Universal Robots URScript: 2024DragonThinMarker_v7.script

def P2024DragonThinMarker_v7():
  step_count_72c97e26_6cb8_45e0_928f_f3c530a1ae50 = 0.0
  thread Step_Counter_Thread_41fc0684_b974_431a_b44c_1ae3c598adf5():
    while (True):
      step_count_72c97e26_6cb8_45e0_928f_f3c530a1ae50 = step_count_72c97e26_6cb8_45e0_928f_f3c530a1ae50 + 1.0
      sync()
    end
  end
  run Step_Counter_Thread_41fc0684_b974_431a_b44c_1ae3c598adf5()
  set_gravity([0.0, 0.0, 9.82])
  set_tcp(p[0.0,0.0,0.0,0.0,0.0,0.0])
  set_standard_analog_input_domain(0, 1)
  set_standard_analog_input_domain(1, 1)
  set_tool_analog_input_domain(0, 1)
  set_tool_analog_input_domain(1, 1)
  set_analog_outputdomain(0, 0)
  set_analog_outputdomain(1, 0)
  set_input_actions_to_default()
  set_target_payload(1.070000, [0.002000, 0.003000, 0.057000], [0.001723, 0.001723, 0.001723, 0.000000, 0.000000, 0.000000])
  set_safety_mode_transition_hardness(1)
  set_tool_communication(True, 1000000, 2, 1, 1.5, 3.5)
  set_tool_output_mode(0)
  set_tool_digital_output_mode(0, 1)
  set_tool_digital_output_mode(1, 1)
  set_tool_voltage(0)
  global Plane_1=p[-0.700006141123905,1.3454883874109249E-6,0.3910559577028425,-1.2089868272251132,-1.2089999932245832,1.20858562628424]
  global Plane_2=p[0.0,0.0,0.0,0.0,0.0,0.0]
  global Point_1=p[0.6913645118948067,-0.12399382748223003,0.49223711947071,-1.2983729986843258,1.1259514972191385,-1.2203503861141718]
  $ 1 "Robot Program"
  $ 2 "Script: polyu_fai_chun_2024.script"
  def Machining1():
    # Default parameters:
    global speed_ms = 0.3
    global speed_rads = 0.75
    global accel_mss = 3
    global accel_radss = 1.2
    global blend_radius_m = 0.001

    # Add subprograms here
    # Start of main program
    # Program generated by RoboDK v5.6.5 for UR10e on 12/01/2024 18:22:17
    # Using nominal kinematics.
    blend_radius_m = 0.000
    speed_ms = 1.000
    # set_reference(p[0.335000, -0.149886, -0.015500, 0.000000, 0.000000, 0.000000])
    set_tcp(p[0.000000, 0.000000, 0.252000, 0.000000, 0.000000, 0.000000])
    # Show Tool
    movej([0.073712, -1.005472, -2.512389, -1.194528, 1.570796, 1.644508],accel_radss,speed_rads,0,blend_radius_m)
    movel([0.073712, -1.005472, -2.512389, -1.194528, 1.570796, 1.644508],accel_mss,speed_ms,0,blend_radius_m)
    # Splitting Linear movement in 6 (instruction 7: MoveL 3)
    movel([0.073712, -1.023685, -2.537003, -1.151700, 1.570796, 1.644508],accel_mss,speed_ms,0,blend_radius_m)
    movel([0.073712, -1.044503, -2.561079, -1.106807, 1.570796, 1.644508],accel_mss,speed_ms,0,blend_radius_m)
    movel([0.073712, -1.068168, -2.584569, -1.059651, 1.570796, 1.644508],accel_mss,speed_ms,0,blend_radius_m)
    movel([0.073712, -1.094942, -2.607420, -1.010026, 1.570796, 1.644508],accel_mss,speed_ms,0,blend_radius_m)
    movel([0.073712, -1.125104, -2.629569, -0.957717, 1.570796, 1.644508],accel_mss,speed_ms,0,blend_radius_m)
    movel([0.073712, -1.158943, -2.650939, -0.902506, 1.570796, 1.644508],accel_mss,speed_ms,0,blend_radius_m)
    movel([0.073712, -1.158943, -2.650939, -0.902506, 1.570796, 1.644508],accel_mss,speed_ms,0,blend_radius_m)
    speed_ms = 1.000
    movel([0.073712, -1.158943, -2.650939, -0.902506, 1.570796, 1.644508],accel_mss,speed_ms,0,blend_radius_m)
    movel([0.073712, -1.158943, -2.650939, -0.902506, 1.570796, 1.644508],accel_mss,speed_ms,0,blend_radius_m)
    movel([0.073712, -1.158943, -2.650939, -0.902506, 1.570796, 1.644508],accel_mss,speed_ms,0,blend_radius_m)
    speed_ms = 0.005
    movel([0.073712, -1.118787, -2.625199, -0.968404, 1.570796, 1.644508],accel_mss,speed_ms,0,blend_radius_m)
    speed_ms = 1.000
    movel([0.073712, -1.158943, -2.650939, -0.902506, 1.570796, 1.644508],accel_mss,speed_ms,0,blend_radius_m)
    speed_ms = 0.040
    movel([0.073712, -1.158943, -2.650939, -0.902506, 1.570796, 1.644508],accel_mss,speed_ms,0,blend_radius_m)
    speed_ms = 1.000
    movel([0.073712, -1.158943, -2.650939, -0.902506, 1.570796, 1.644508],accel_mss,speed_ms,0,blend_radius_m)
    # Splitting Linear movement in 4 (instruction 21: MoveL 12)
    movel([0.101880, -1.181857, -2.640286, -0.890246, 1.570796, 1.672676],accel_mss,speed_ms,0,blend_radius_m)
    movel([0.128207, -1.205564, -2.628681, -0.878144, 1.570796, 1.699004],accel_mss,speed_ms,0,blend_radius_m)
    movel([0.152802, -1.229857, -2.616150, -0.866382, 1.570796, 1.723598],accel_mss,speed_ms,0,blend_radius_m)
    movel([0.175774, -1.254553, -2.602722, -0.855114, 1.570796, 1.746570],accel_mss,speed_ms,0,blend_radius_m)
    speed_ms = 0.005
    movel([0.175774, -1.298704, -2.625119, -0.788567, 1.570796, 1.746570],accel_mss,speed_ms,0,blend_radius_m)
    speed_ms = 0.025
    movel([0.175467, -1.296515, -2.626415, -0.789459, 1.570796, 1.746263],accel_mss,speed_ms,0,blend_radius_m)
    movel([0.175132, -1.295590, -2.626961, -0.789837, 1.570796, 1.745929],accel_mss,speed_ms,0,blend_radius_m)
    movel([0.174656, -1.294762, -2.627449, -0.790178, 1.570796, 1.745452],accel_mss,speed_ms,0,blend_radius_m)
    movel([0.174050, -1.294049, -2.627869, -0.790471, 1.570796, 1.744846],accel_mss,speed_ms,0,blend_radius_m)
    movel([0.173318, -1.293452, -2.628219, -0.790718, 1.570796, 1.744114],accel_mss,speed_ms,0,blend_radius_m)
    movel([0.172433, -1.292952, -2.628513, -0.790925, 1.570796, 1.743230],accel_mss,speed_ms,0,blend_radius_m)
    movel([0.171452, -1.292568, -2.628738, -0.791083, 1.570796, 1.742248],accel_mss,speed_ms,0,blend_radius_m)
    movel([0.169238, -1.292109, -2.629007, -0.791274, 1.570796, 1.740034],accel_mss,speed_ms,0,blend_radius_m)
    movel([0.166824, -1.292044, -2.629045, -0.791300, 1.570796, 1.737621],accel_mss,speed_ms,0,blend_radius_m)
    movel([0.164077, -1.292380, -2.628848, -0.791161, 1.570796, 1.734873],accel_mss,speed_ms,0,blend_radius_m)
    movel([0.160852, -1.293136, -2.628405, -0.790848, 1.570796, 1.731649],accel_mss,speed_ms,0,blend_radius_m)
    movel([0.158343, -1.293899, -2.627957, -0.790533, 1.570796, 1.729139],accel_mss,speed_ms,0,blend_radius_m)
    movel([0.156195, -1.294698, -2.627487, -0.790204, 1.570796, 1.726992],accel_mss,speed_ms,0,blend_radius_m)
    movel([0.154013, -1.295690, -2.626903, -0.789797, 1.570796, 1.724809],accel_mss,speed_ms,0,blend_radius_m)
    movel([0.151400, -1.297044, -2.626103, -0.789243, 1.570796, 1.722196],accel_mss,speed_ms,0,blend_radius_m)
    movel([0.148354, -1.298788, -2.625069, -0.788532, 1.570796, 1.719150],accel_mss,speed_ms,0,blend_radius_m)
    movel([0.140219, -1.303870, -2.622034, -0.786485, 1.570796, 1.711015],accel_mss,speed_ms,0,blend_radius_m)
    movel([0.140032, -1.304046, -2.621928, -0.786415, 1.570796, 1.710829],accel_mss,speed_ms,0,blend_radius_m)
    movel([0.139940, -1.304251, -2.621805, -0.786333, 1.570796, 1.710737],accel_mss,speed_ms,0,blend_radius_m)
    movel([0.140046, -1.304840, -2.621451, -0.786098, 1.570796, 1.710842],accel_mss,speed_ms,0,blend_radius_m)
    movel([0.143328, -1.309440, -2.618669, -0.784280, 1.570796, 1.714124],accel_mss,speed_ms,0,blend_radius_m)
    movel([0.145350, -1.311978, -2.617122, -0.783289, 1.570796, 1.716147],accel_mss,speed_ms,0,blend_radius_m)
    movel([0.153033, -1.320929, -2.611599, -0.779860, 1.570796, 1.723829],accel_mss,speed_ms,0,blend_radius_m)
    movel([0.157376, -1.325880, -2.608499, -0.778010, 1.570796, 1.728172],accel_mss,speed_ms,0,blend_radius_m)
    movel([0.160651, -1.329420, -2.606262, -0.776707, 1.570796, 1.731447],accel_mss,speed_ms,0,blend_radius_m)
    movel([0.161108, -1.329847, -2.605991, -0.776551, 1.570796, 1.731904],accel_mss,speed_ms,0,blend_radius_m)
    movel([0.161761, -1.330342, -2.605676, -0.776371, 1.570796, 1.732557],accel_mss,speed_ms,0,blend_radius_m)
    movel([0.162354, -1.330373, -2.605656, -0.776359, 1.570796, 1.733150],accel_mss,speed_ms,0,blend_radius_m)
    movel([0.162959, -1.330023, -2.605879, -0.776487, 1.570796, 1.733755],accel_mss,speed_ms,0,blend_radius_m)
    movel([0.163738, -1.329104, -2.606462, -0.776823, 1.570796, 1.734534],accel_mss,speed_ms,0,blend_radius_m)
    movel([0.165104, -1.327071, -2.607748, -0.777570, 1.570796, 1.735901],accel_mss,speed_ms,0,blend_radius_m)
    movel([0.167659, -1.322835, -2.610409, -0.779144, 1.570796, 1.738455],accel_mss,speed_ms,0,blend_radius_m)
    movel([0.169919, -1.318408, -2.613166, -0.780815, 1.570796, 1.740716],accel_mss,speed_ms,0,blend_radius_m)
    movel([0.171903, -1.313743, -2.616042, -0.782604, 1.570796, 1.742699],accel_mss,speed_ms,0,blend_radius_m)
    movel([0.173625, -1.308797, -2.619060, -0.784532, 1.570796, 1.744421],accel_mss,speed_ms,0,blend_radius_m)
    movel([0.174404, -1.306055, -2.620719, -0.785615, 1.570796, 1.745200],accel_mss,speed_ms,0,blend_radius_m)
    movel([0.175649, -1.300261, -2.624193, -0.787936, 1.570796, 1.746445],accel_mss,speed_ms,0,blend_radius_m)
    movel([0.175774, -1.298704, -2.625119, -0.788567, 1.570796, 1.746570],accel_mss,speed_ms,0,blend_radius_m)
    movel([0.175467, -1.296515, -2.626415, -0.789459, 1.570796, 1.746263],accel_mss,speed_ms,0,blend_radius_m)
    speed_ms = 0.005
    movel([0.175467, -1.287281, -2.622040, -0.803067, 1.570796, 1.746263],accel_mss,speed_ms,0,blend_radius_m)
    speed_ms = 0.040
    movel([0.174810, -1.299280, -2.614952, -0.798157, 1.570796, 1.745606],accel_mss,speed_ms,0,blend_radius_m)
    speed_ms = 0.005
    movel([0.174810, -1.308444, -2.619274, -0.784671, 1.570796, 1.745606],accel_mss,speed_ms,0,blend_radius_m)
    speed_ms = 0.025
    movel([0.172959, -1.313681, -2.616080, -0.782628, 1.570796, 1.743756],accel_mss,speed_ms,0,blend_radius_m)
    movel([0.171021, -1.318273, -2.613249, -0.780867, 1.570796, 1.741817],accel_mss,speed_ms,0,blend_radius_m)
    movel([0.168851, -1.322542, -2.610593, -0.779254, 1.570796, 1.739648],accel_mss,speed_ms,0,blend_radius_m)
    movel([0.166314, -1.326792, -2.607924, -0.777673, 1.570796, 1.737110],accel_mss,speed_ms,0,blend_radius_m)
    movel([0.163959, -1.330191, -2.605772, -0.776426, 1.570796, 1.734756],accel_mss,speed_ms,0,blend_radius_m)
    movel([0.163273, -1.330890, -2.605328, -0.776171, 1.570796, 1.734070],accel_mss,speed_ms,0,blend_radius_m)
    movel([0.162439, -1.331386, -2.605012, -0.775991, 1.570796, 1.733235],accel_mss,speed_ms,0,blend_radius_m)
    movel([0.161654, -1.331560, -2.604902, -0.775928, 1.570796, 1.732450],accel_mss,speed_ms,0,blend_radius_m)
    movel([0.161027, -1.331383, -2.605014, -0.775992, 1.570796, 1.731824],accel_mss,speed_ms,0,blend_radius_m)
    movel([0.159182, -1.329800, -2.606021, -0.776568, 1.570796, 1.729978],accel_mss,speed_ms,0,blend_radius_m)
    movel([0.154933, -1.325131, -2.608970, -0.778288, 1.570796, 1.725729],accel_mss,speed_ms,0,blend_radius_m)
    movel([0.149543, -1.318950, -2.612830, -0.780609, 1.570796, 1.720340],accel_mss,speed_ms,0,blend_radius_m)
    movel([0.144364, -1.312895, -2.616561, -0.782932, 1.570796, 1.715160],accel_mss,speed_ms,0,blend_radius_m)
    movel([0.141237, -1.308969, -2.618955, -0.784465, 1.570796, 1.712033],accel_mss,speed_ms,0,blend_radius_m)
    movel([0.139694, -1.306790, -2.620275, -0.785324, 1.570796, 1.710491],accel_mss,speed_ms,0,blend_radius_m)
    movel([0.138982, -1.305403, -2.621112, -0.785874, 1.570796, 1.709778],accel_mss,speed_ms,0,blend_radius_m)
    movel([0.138836, -1.304410, -2.621710, -0.786270, 1.570796, 1.709632],accel_mss,speed_ms,0,blend_radius_m)
    movel([0.138954, -1.304019, -2.621945, -0.786426, 1.570796, 1.709750],accel_mss,speed_ms,0,blend_radius_m)
    movel([0.139242, -1.303642, -2.622171, -0.786576, 1.570796, 1.710039],accel_mss,speed_ms,0,blend_radius_m)
    movel([0.139895, -1.303121, -2.622483, -0.786785, 1.570796, 1.710691],accel_mss,speed_ms,0,blend_radius_m)
    movel([0.145279, -1.299642, -2.624561, -0.788186, 1.570796, 1.716076],accel_mss,speed_ms,0,blend_radius_m)
    movel([0.147733, -1.298138, -2.625454, -0.788797, 1.570796, 1.718530],accel_mss,speed_ms,0,blend_radius_m)
    movel([0.150828, -1.296376, -2.626497, -0.789515, 1.570796, 1.721624],accel_mss,speed_ms,0,blend_radius_m)
    movel([0.153961, -1.294776, -2.627441, -0.790172, 1.570796, 1.724758],accel_mss,speed_ms,0,blend_radius_m)
    movel([0.156801, -1.293517, -2.628181, -0.790691, 1.570796, 1.727598],accel_mss,speed_ms,0,blend_radius_m)
    movel([0.159642, -1.292475, -2.628792, -0.791122, 1.570796, 1.730438],accel_mss,speed_ms,0,blend_radius_m)
    movel([0.162247, -1.291733, -2.629227, -0.791430, 1.570796, 1.733043],accel_mss,speed_ms,0,blend_radius_m)
    movel([0.164801, -1.291232, -2.629519, -0.791638, 1.570796, 1.735598],accel_mss,speed_ms,0,blend_radius_m)
    movel([0.167190, -1.290996, -2.629657, -0.791736, 1.570796, 1.737986],accel_mss,speed_ms,0,blend_radius_m)
    movel([0.169469, -1.291023, -2.629641, -0.791725, 1.570796, 1.740266],accel_mss,speed_ms,0,blend_radius_m)
    movel([0.171128, -1.291248, -2.629510, -0.791631, 1.570796, 1.741924],accel_mss,speed_ms,0,blend_radius_m)
    movel([0.172657, -1.291674, -2.629261, -0.791454, 1.570796, 1.743454],accel_mss,speed_ms,0,blend_radius_m)
    movel([0.173914, -1.292270, -2.628912, -0.791207, 1.570796, 1.744711],accel_mss,speed_ms,0,blend_radius_m)
    movel([0.174977, -1.293079, -2.628438, -0.790872, 1.570796, 1.745773],accel_mss,speed_ms,0,blend_radius_m)
    movel([0.175808, -1.294073, -2.627854, -0.790461, 1.570796, 1.746605],accel_mss,speed_ms,0,blend_radius_m)
    movel([0.176410, -1.295244, -2.627165, -0.789980, 1.570796, 1.747207],accel_mss,speed_ms,0,blend_radius_m)
    movel([0.176810, -1.296630, -2.626347, -0.789412, 1.570796, 1.747606],accel_mss,speed_ms,0,blend_radius_m)
    movel([0.176990, -1.298135, -2.625456, -0.788798, 1.570796, 1.747786],accel_mss,speed_ms,0,blend_radius_m)
    movel([0.176880, -1.299644, -2.624560, -0.788185, 1.570796, 1.747676],accel_mss,speed_ms,0,blend_radius_m)
    movel([0.176287, -1.302678, -2.622749, -0.786962, 1.570796, 1.747084],accel_mss,speed_ms,0,blend_radius_m)
    movel([0.175547, -1.305881, -2.620824, -0.785684, 1.570796, 1.746344],accel_mss,speed_ms,0,blend_radius_m)
    movel([0.174810, -1.308444, -2.619274, -0.784671, 1.570796, 1.745606],accel_mss,speed_ms,0,blend_radius_m)
    movel([0.173912, -1.310987, -2.617727, -0.783675, 1.570796, 1.744708],accel_mss,speed_ms,0,blend_radius_m)
    speed_ms = 0.005
    movel([0.173912, -1.301837, -2.613417, -0.797134, 1.570796, 1.744708],accel_mss,speed_ms,0,blend_radius_m)
    speed_ms = 0.040
    # Splitting Linear movement in 4 (instruction 117: MoveL 100)
    movel([0.163813, -1.329309, -2.596395, -0.786686, 1.570796, 1.734610],accel_mss,speed_ms,0,blend_radius_m)
    movel([0.154297, -1.355614, -2.579147, -0.777628, 1.570796, 1.725093],accel_mss,speed_ms,0,blend_radius_m)
    movel([0.145312, -1.380862, -2.561692, -0.769834, 1.570796, 1.716108],accel_mss,speed_ms,0,blend_radius_m)
    movel([0.136812, -1.405151, -2.544044, -0.763194, 1.570796, 1.707609],accel_mss,speed_ms,0,blend_radius_m)
    speed_ms = 0.005
    movel([0.136812, -1.413611, -2.547901, -0.750877, 1.570796, 1.707609],accel_mss,speed_ms,0,blend_radius_m)
    speed_ms = 0.025
    movel([0.136960, -1.413086, -2.548297, -0.751006, 1.570796, 1.707756],accel_mss,speed_ms,0,blend_radius_m)
    movel([0.137280, -1.410569, -2.550188, -0.751632, 1.570796, 1.708076],accel_mss,speed_ms,0,blend_radius_m)
    movel([0.137084, -1.408675, -2.551604, -0.752109, 1.570796, 1.707880],accel_mss,speed_ms,0,blend_radius_m)
    movel([0.136478, -1.406567, -2.553175, -0.752647, 1.570796, 1.707274],accel_mss,speed_ms,0,blend_radius_m)
    movel([0.135486, -1.404266, -2.554882, -0.753241, 1.570796, 1.706282],accel_mss,speed_ms,0,blend_radius_m)
    movel([0.134091, -1.401787, -2.556712, -0.753889, 1.570796, 1.704888],accel_mss,speed_ms,0,blend_radius_m)
    movel([0.133438, -1.400815, -2.557428, -0.754146, 1.570796, 1.704235],accel_mss,speed_ms,0,blend_radius_m)
    movel([0.132951, -1.400309, -2.557799, -0.754280, 1.570796, 1.703748],accel_mss,speed_ms,0,blend_radius_m)
    movel([0.132501, -1.400110, -2.557946, -0.754333, 1.570796, 1.703298],accel_mss,speed_ms,0,blend_radius_m)
    movel([0.132010, -1.400164, -2.557906, -0.754319, 1.570796, 1.702806],accel_mss,speed_ms,0,blend_radius_m)
    movel([0.131521, -1.400467, -2.557683, -0.754238, 1.570796, 1.702317],accel_mss,speed_ms,0,blend_radius_m)
    movel([0.131266, -1.400883, -2.557378, -0.754128, 1.570796, 1.702062],accel_mss,speed_ms,0,blend_radius_m)
    movel([0.131373, -1.401180, -2.557160, -0.754050, 1.570796, 1.702169],accel_mss,speed_ms,0,blend_radius_m)
    movel([0.132162, -1.401260, -2.557101, -0.754029, 1.570796, 1.702958],accel_mss,speed_ms,0,blend_radius_m)
    movel([0.132555, -1.401611, -2.556842, -0.753936, 1.570796, 1.703352],accel_mss,speed_ms,0,blend_radius_m)
    movel([0.134004, -1.403943, -2.555121, -0.753325, 1.570796, 1.704800],accel_mss,speed_ms,0,blend_radius_m)
    movel([0.135071, -1.406059, -2.553553, -0.752777, 1.570796, 1.705868],accel_mss,speed_ms,0,blend_radius_m)
    movel([0.135785, -1.408024, -2.552090, -0.752275, 1.570796, 1.706581],accel_mss,speed_ms,0,blend_radius_m)
    movel([0.136159, -1.409851, -2.550725, -0.751812, 1.570796, 1.706955],accel_mss,speed_ms,0,blend_radius_m)
    movel([0.136189, -1.411547, -2.549454, -0.751388, 1.570796, 1.706985],accel_mss,speed_ms,0,blend_radius_m)
    movel([0.136087, -1.412720, -2.548572, -0.751097, 1.570796, 1.706884],accel_mss,speed_ms,0,blend_radius_m)
    movel([0.135567, -1.411763, -2.549291, -0.751334, 1.570796, 1.706364],accel_mss,speed_ms,0,blend_radius_m)
    movel([0.134960, -1.410840, -2.549984, -0.751564, 1.570796, 1.705756],accel_mss,speed_ms,0,blend_radius_m)
    movel([0.134201, -1.410029, -2.550592, -0.751768, 1.570796, 1.704998],accel_mss,speed_ms,0,blend_radius_m)
    movel([0.133183, -1.409207, -2.551207, -0.751975, 1.570796, 1.703979],accel_mss,speed_ms,0,blend_radius_m)
    movel([0.132066, -1.408483, -2.551748, -0.752158, 1.570796, 1.702862],accel_mss,speed_ms,0,blend_radius_m)
    movel([0.130773, -1.407814, -2.552247, -0.752328, 1.570796, 1.701569],accel_mss,speed_ms,0,blend_radius_m)
    movel([0.129389, -1.407256, -2.552662, -0.752470, 1.570796, 1.700185],accel_mss,speed_ms,0,blend_radius_m)
    movel([0.127928, -1.406809, -2.552995, -0.752585, 1.570796, 1.698724],accel_mss,speed_ms,0,blend_radius_m)
    movel([0.126392, -1.406478, -2.553242, -0.752670, 1.570796, 1.697188],accel_mss,speed_ms,0,blend_radius_m)
    movel([0.124687, -1.406237, -2.553421, -0.752732, 1.570796, 1.695483],accel_mss,speed_ms,0,blend_radius_m)
    movel([0.123487, -1.406221, -2.553432, -0.752735, 1.570796, 1.694283],accel_mss,speed_ms,0,blend_radius_m)
    movel([0.122540, -1.406414, -2.553289, -0.752686, 1.570796, 1.693336],accel_mss,speed_ms,0,blend_radius_m)
    movel([0.121683, -1.406830, -2.552980, -0.752579, 1.570796, 1.692479],accel_mss,speed_ms,0,blend_radius_m)
    movel([0.121218, -1.407199, -2.552705, -0.752485, 1.570796, 1.692014],accel_mss,speed_ms,0,blend_radius_m)
    movel([0.120891, -1.407598, -2.552408, -0.752383, 1.570796, 1.691687],accel_mss,speed_ms,0,blend_radius_m)
    movel([0.120677, -1.408078, -2.552050, -0.752261, 1.570796, 1.691473],accel_mss,speed_ms,0,blend_radius_m)
    movel([0.120519, -1.409292, -2.551143, -0.751953, 1.570796, 1.691315],accel_mss,speed_ms,0,blend_radius_m)
    movel([0.120597, -1.410164, -2.550491, -0.751734, 1.570796, 1.691393],accel_mss,speed_ms,0,blend_radius_m)
    movel([0.120924, -1.411776, -2.549282, -0.751331, 1.570796, 1.691721],accel_mss,speed_ms,0,blend_radius_m)
    movel([0.120137, -1.411178, -2.549731, -0.751480, 1.570796, 1.690933],accel_mss,speed_ms,0,blend_radius_m)
    movel([0.119142, -1.410325, -2.550371, -0.751693, 1.570796, 1.689938],accel_mss,speed_ms,0,blend_radius_m)
    movel([0.118017, -1.409589, -2.550922, -0.751879, 1.570796, 1.688813],accel_mss,speed_ms,0,blend_radius_m)
    movel([0.116588, -1.408871, -2.551458, -0.752060, 1.570796, 1.687384],accel_mss,speed_ms,0,blend_radius_m)
    movel([0.114638, -1.408066, -2.552059, -0.752264, 1.570796, 1.685434],accel_mss,speed_ms,0,blend_radius_m)
    movel([0.110959, -1.406603, -2.553148, -0.752637, 1.570796, 1.681756],accel_mss,speed_ms,0,blend_radius_m)
    movel([0.108642, -1.405547, -2.553933, -0.752909, 1.570796, 1.679439],accel_mss,speed_ms,0,blend_radius_m)
    movel([0.106996, -1.404575, -2.554653, -0.753160, 1.570796, 1.677792],accel_mss,speed_ms,0,blend_radius_m)
    movel([0.105601, -1.403457, -2.555480, -0.753451, 1.570796, 1.676397],accel_mss,speed_ms,0,blend_radius_m)
    movel([0.105049, -1.402986, -2.555828, -0.753574, 1.570796, 1.675845],accel_mss,speed_ms,0,blend_radius_m)
    movel([0.104656, -1.402804, -2.555963, -0.753622, 1.570796, 1.675452],accel_mss,speed_ms,0,blend_radius_m)
    movel([0.104367, -1.402858, -2.555923, -0.753608, 1.570796, 1.675163],accel_mss,speed_ms,0,blend_radius_m)
    movel([0.104133, -1.403095, -2.555748, -0.753546, 1.570796, 1.674929],accel_mss,speed_ms,0,blend_radius_m)
    movel([0.104093, -1.403268, -2.555620, -0.753501, 1.570796, 1.674889],accel_mss,speed_ms,0,blend_radius_m)
    movel([0.104524, -1.406129, -2.553501, -0.752759, 1.570796, 1.675320],accel_mss,speed_ms,0,blend_radius_m)
    movel([0.104631, -1.406790, -2.553009, -0.752590, 1.570796, 1.675427],accel_mss,speed_ms,0,blend_radius_m)
    movel([0.104692, -1.407427, -2.552536, -0.752427, 1.570796, 1.675488],accel_mss,speed_ms,0,blend_radius_m)
    movel([0.102290, -1.405992, -2.553602, -0.752794, 1.570796, 1.673087],accel_mss,speed_ms,0,blend_radius_m)
    movel([0.100620, -1.404841, -2.554457, -0.753092, 1.570796, 1.671417],accel_mss,speed_ms,0,blend_radius_m)
    movel([0.099425, -1.403815, -2.555216, -0.753358, 1.570796, 1.670222],accel_mss,speed_ms,0,blend_radius_m)
    movel([0.098377, -1.402613, -2.556104, -0.753672, 1.570796, 1.669174],accel_mss,speed_ms,0,blend_radius_m)
    movel([0.095814, -1.399011, -2.558752, -0.754627, 1.570796, 1.666610],accel_mss,speed_ms,0,blend_radius_m)
    movel([0.094727, -1.397866, -2.559589, -0.754934, 1.570796, 1.665523],accel_mss,speed_ms,0,blend_radius_m)
    movel([0.093735, -1.397245, -2.560043, -0.755101, 1.570796, 1.664531],accel_mss,speed_ms,0,blend_radius_m)
    movel([0.093259, -1.397104, -2.560145, -0.755139, 1.570796, 1.664056],accel_mss,speed_ms,0,blend_radius_m)
    movel([0.092715, -1.397075, -2.560166, -0.755147, 1.570796, 1.663511],accel_mss,speed_ms,0,blend_radius_m)
    movel([0.092023, -1.397198, -2.560077, -0.755114, 1.570796, 1.662819],accel_mss,speed_ms,0,blend_radius_m)
    movel([0.091298, -1.397494, -2.559861, -0.755034, 1.570796, 1.662095],accel_mss,speed_ms,0,blend_radius_m)
    movel([0.090566, -1.397956, -2.559523, -0.754910, 1.570796, 1.661362],accel_mss,speed_ms,0,blend_radius_m)
    movel([0.089095, -1.399249, -2.558577, -0.754563, 1.570796, 1.659892],accel_mss,speed_ms,0,blend_radius_m)
    movel([0.088807, -1.398175, -2.559363, -0.754851, 1.570796, 1.659604],accel_mss,speed_ms,0,blend_radius_m)
    movel([0.088677, -1.397590, -2.559790, -0.755008, 1.570796, 1.659474],accel_mss,speed_ms,0,blend_radius_m)
    movel([0.086678, -1.390759, -2.564745, -0.756884, 1.570796, 1.657474],accel_mss,speed_ms,0,blend_radius_m)
    movel([0.086361, -1.389318, -2.565782, -0.757289, 1.570796, 1.657158],accel_mss,speed_ms,0,blend_radius_m)
    movel([0.086303, -1.388031, -2.566706, -0.757652, 1.570796, 1.657099],accel_mss,speed_ms,0,blend_radius_m)
    movel([0.086463, -1.385965, -2.568183, -0.758241, 1.570796, 1.657259],accel_mss,speed_ms,0,blend_radius_m)
    movel([0.086845, -1.383220, -2.570135, -0.759033, 1.570796, 1.657641],accel_mss,speed_ms,0,blend_radius_m)
    movel([0.087125, -1.382255, -2.570820, -0.759315, 1.570796, 1.657921],accel_mss,speed_ms,0,blend_radius_m)
    movel([0.088538, -1.378520, -2.573454, -0.760415, 1.570796, 1.659334],accel_mss,speed_ms,0,blend_radius_m)
    movel([0.088847, -1.377865, -2.573914, -0.760610, 1.570796, 1.659643],accel_mss,speed_ms,0,blend_radius_m)
    movel([0.089252, -1.377361, -2.574268, -0.760760, 1.570796, 1.660049],accel_mss,speed_ms,0,blend_radius_m)
    movel([0.089322, -1.377088, -2.574459, -0.760842, 1.570796, 1.660119],accel_mss,speed_ms,0,blend_radius_m)
    movel([0.089228, -1.376863, -2.574617, -0.760909, 1.570796, 1.660025],accel_mss,speed_ms,0,blend_radius_m)
    movel([0.088991, -1.376732, -2.574708, -0.760949, 1.570796, 1.659787],accel_mss,speed_ms,0,blend_radius_m)
    movel([0.088772, -1.376745, -2.574699, -0.760945, 1.570796, 1.659568],accel_mss,speed_ms,0,blend_radius_m)
    movel([0.088542, -1.376869, -2.574612, -0.760908, 1.570796, 1.659338],accel_mss,speed_ms,0,blend_radius_m)
    movel([0.088083, -1.377390, -2.574248, -0.760752, 1.570796, 1.658880],accel_mss,speed_ms,0,blend_radius_m)
    movel([0.087563, -1.378426, -2.573520, -0.760443, 1.570796, 1.658359],accel_mss,speed_ms,0,blend_radius_m)
    movel([0.086135, -1.382410, -2.570710, -0.759269, 1.570796, 1.656932],accel_mss,speed_ms,0,blend_radius_m)
    movel([0.085693, -1.383923, -2.569636, -0.758830, 1.570796, 1.656489],accel_mss,speed_ms,0,blend_radius_m)
    movel([0.085220, -1.386694, -2.567662, -0.758033, 1.570796, 1.656017],accel_mss,speed_ms,0,blend_radius_m)
    movel([0.085156, -1.388244, -2.566553, -0.757592, 1.570796, 1.655952],accel_mss,speed_ms,0,blend_radius_m)
    movel([0.085288, -1.389626, -2.565561, -0.757202, 1.570796, 1.656084],accel_mss,speed_ms,0,blend_radius_m)
    movel([0.085687, -1.391336, -2.564330, -0.756723, 1.570796, 1.656483],accel_mss,speed_ms,0,blend_radius_m)
    movel([0.087127, -1.396101, -2.560877, -0.755411, 1.570796, 1.657923],accel_mss,speed_ms,0,blend_radius_m)
    movel([0.087508, -1.397558, -2.559814, -0.755017, 1.570796, 1.658304],accel_mss,speed_ms,0,blend_radius_m)
    movel([0.088079, -1.400709, -2.557506, -0.754174, 1.570796, 1.658875],accel_mss,speed_ms,0,blend_radius_m)
    movel([0.088230, -1.401088, -2.557227, -0.754074, 1.570796, 1.659026],accel_mss,speed_ms,0,blend_radius_m)
    movel([0.088515, -1.401157, -2.557177, -0.754056, 1.570796, 1.659311],accel_mss,speed_ms,0,blend_radius_m)
    movel([0.088888, -1.400924, -2.557347, -0.754117, 1.570796, 1.659684],accel_mss,speed_ms,0,blend_radius_m)
    movel([0.089305, -1.400387, -2.557742, -0.754260, 1.570796, 1.660101],accel_mss,speed_ms,0,blend_radius_m)
    movel([0.089783, -1.399740, -2.558217, -0.754432, 1.570796, 1.660580],accel_mss,speed_ms,0,blend_radius_m)
    movel([0.090394, -1.399084, -2.558698, -0.754607, 1.570796, 1.661191],accel_mss,speed_ms,0,blend_radius_m)
    movel([0.091027, -1.398524, -2.559108, -0.754757, 1.570796, 1.661823],accel_mss,speed_ms,0,blend_radius_m)
    movel([0.091557, -1.398188, -2.559353, -0.754847, 1.570796, 1.662354],accel_mss,speed_ms,0,blend_radius_m)
    movel([0.092171, -1.398032, -2.559468, -0.754889, 1.570796, 1.662968],accel_mss,speed_ms,0,blend_radius_m)
    movel([0.092861, -1.398118, -2.559405, -0.754866, 1.570796, 1.663658],accel_mss,speed_ms,0,blend_radius_m)
    movel([0.093562, -1.398429, -2.559178, -0.754783, 1.570796, 1.664359],accel_mss,speed_ms,0,blend_radius_m)
    movel([0.094200, -1.398945, -2.558800, -0.754644, 1.570796, 1.664996],accel_mss,speed_ms,0,blend_radius_m)
    movel([0.094561, -1.399351, -2.558502, -0.754536, 1.570796, 1.665357],accel_mss,speed_ms,0,blend_radius_m)
    movel([0.098013, -1.404105, -2.555001, -0.753283, 1.570796, 1.668809],accel_mss,speed_ms,0,blend_radius_m)
    movel([0.098347, -1.404499, -2.554710, -0.753180, 1.570796, 1.669143],accel_mss,speed_ms,0,blend_radius_m)
    movel([0.099589, -1.405494, -2.553973, -0.752923, 1.570796, 1.670385],accel_mss,speed_ms,0,blend_radius_m)
    movel([0.100597, -1.406207, -2.553443, -0.752739, 1.570796, 1.671393],accel_mss,speed_ms,0,blend_radius_m)
    movel([0.105149, -1.409357, -2.551095, -0.751937, 1.570796, 1.675945],accel_mss,speed_ms,0,blend_radius_m)
    movel([0.106031, -1.410013, -2.550605, -0.751772, 1.570796, 1.676827],accel_mss,speed_ms,0,blend_radius_m)
    movel([0.106225, -1.410030, -2.550591, -0.751767, 1.570796, 1.677021],accel_mss,speed_ms,0,blend_radius_m)
    movel([0.106437, -1.409903, -2.550687, -0.751800, 1.570796, 1.677233],accel_mss,speed_ms,0,blend_radius_m)
    movel([0.106593, -1.409667, -2.550863, -0.751859, 1.570796, 1.677389],accel_mss,speed_ms,0,blend_radius_m)
    movel([0.106611, -1.409441, -2.551033, -0.751916, 1.570796, 1.677408],accel_mss,speed_ms,0,blend_radius_m)
    movel([0.105600, -1.405987, -2.553606, -0.752796, 1.570796, 1.676396],accel_mss,speed_ms,0,blend_radius_m)
    movel([0.105382, -1.404992, -2.554345, -0.753053, 1.570796, 1.676178],accel_mss,speed_ms,0,blend_radius_m)
    movel([0.107701, -1.406321, -2.553358, -0.752710, 1.570796, 1.678497],accel_mss,speed_ms,0,blend_radius_m)
    movel([0.109036, -1.406958, -2.552884, -0.752547, 1.570796, 1.679832],accel_mss,speed_ms,0,blend_radius_m)
    movel([0.112944, -1.408534, -2.551710, -0.752145, 1.570796, 1.683740],accel_mss,speed_ms,0,blend_radius_m)
    movel([0.115927, -1.409742, -2.550807, -0.751840, 1.570796, 1.686724],accel_mss,speed_ms,0,blend_radius_m)
    movel([0.117594, -1.410633, -2.550139, -0.751616, 1.570796, 1.688391],accel_mss,speed_ms,0,blend_radius_m)
    movel([0.119035, -1.411772, -2.549285, -0.751332, 1.570796, 1.689831],accel_mss,speed_ms,0,blend_radius_m)
    movel([0.121575, -1.414285, -2.547393, -0.750712, 1.570796, 1.692371],accel_mss,speed_ms,0,blend_radius_m)
    movel([0.121884, -1.414519, -2.547215, -0.750654, 1.570796, 1.692680],accel_mss,speed_ms,0,blend_radius_m)
    movel([0.122364, -1.414644, -2.547121, -0.750624, 1.570796, 1.693160],accel_mss,speed_ms,0,blend_radius_m)
    movel([0.122659, -1.414449, -2.547268, -0.750671, 1.570796, 1.693456],accel_mss,speed_ms,0,blend_radius_m)
    movel([0.122786, -1.414128, -2.547511, -0.750750, 1.570796, 1.693583],accel_mss,speed_ms,0,blend_radius_m)
    movel([0.122715, -1.413570, -2.547932, -0.750887, 1.570796, 1.693512],accel_mss,speed_ms,0,blend_radius_m)
    movel([0.121659, -1.410088, -2.550548, -0.751753, 1.570796, 1.692455],accel_mss,speed_ms,0,blend_radius_m)
    movel([0.121446, -1.409090, -2.551295, -0.752004, 1.570796, 1.692242],accel_mss,speed_ms,0,blend_radius_m)
    movel([0.121439, -1.408575, -2.551679, -0.752135, 1.570796, 1.692235],accel_mss,speed_ms,0,blend_radius_m)
    movel([0.121484, -1.408388, -2.551819, -0.752182, 1.570796, 1.692280],accel_mss,speed_ms,0,blend_radius_m)
    movel([0.121829, -1.407746, -2.552297, -0.752345, 1.570796, 1.692625],accel_mss,speed_ms,0,blend_radius_m)
    movel([0.122077, -1.407507, -2.552476, -0.752406, 1.570796, 1.692873],accel_mss,speed_ms,0,blend_radius_m)
    movel([0.122378, -1.407341, -2.552599, -0.752449, 1.570796, 1.693174],accel_mss,speed_ms,0,blend_radius_m)
    movel([0.123206, -1.407142, -2.552748, -0.752500, 1.570796, 1.694002],accel_mss,speed_ms,0,blend_radius_m)
    movel([0.124336, -1.407146, -2.552745, -0.752499, 1.570796, 1.695133],accel_mss,speed_ms,0,blend_radius_m)
    movel([0.125835, -1.407372, -2.552576, -0.752441, 1.570796, 1.696631],accel_mss,speed_ms,0,blend_radius_m)
    movel([0.127408, -1.407740, -2.552302, -0.752347, 1.570796, 1.698205],accel_mss,speed_ms,0,blend_radius_m)
    movel([0.128900, -1.408223, -2.551942, -0.752224, 1.570796, 1.699697],accel_mss,speed_ms,0,blend_radius_m)
    movel([0.130280, -1.408803, -2.551509, -0.752077, 1.570796, 1.701076],accel_mss,speed_ms,0,blend_radius_m)
    movel([0.131564, -1.409495, -2.550992, -0.751902, 1.570796, 1.702360],accel_mss,speed_ms,0,blend_radius_m)
    movel([0.132655, -1.410231, -2.550441, -0.751717, 1.570796, 1.703451],accel_mss,speed_ms,0,blend_radius_m)
    movel([0.133637, -1.411071, -2.549812, -0.751507, 1.570796, 1.704434],accel_mss,speed_ms,0,blend_radius_m)
    movel([0.134359, -1.411893, -2.549194, -0.751302, 1.570796, 1.705155],accel_mss,speed_ms,0,blend_radius_m)
    movel([0.134925, -1.412833, -2.548487, -0.751069, 1.570796, 1.705721],accel_mss,speed_ms,0,blend_radius_m)
    movel([0.135624, -1.413985, -2.547619, -0.750785, 1.570796, 1.706420],accel_mss,speed_ms,0,blend_radius_m)
    movel([0.135916, -1.414180, -2.547472, -0.750737, 1.570796, 1.706712],accel_mss,speed_ms,0,blend_radius_m)
    movel([0.136439, -1.414124, -2.547514, -0.750751, 1.570796, 1.707235],accel_mss,speed_ms,0,blend_radius_m)
    movel([0.136587, -1.414019, -2.547593, -0.750777, 1.570796, 1.707383],accel_mss,speed_ms,0,blend_radius_m)
    movel([0.136812, -1.413611, -2.547901, -0.750877, 1.570796, 1.707609],accel_mss,speed_ms,0,blend_radius_m)
    movel([0.136960, -1.413086, -2.548297, -0.751006, 1.570796, 1.707756],accel_mss,speed_ms,0,blend_radius_m)
    movel([0.137159, -1.411521, -2.549473, -0.751394, 1.570796, 1.707955],accel_mss,speed_ms,0,blend_radius_m)
    speed_ms = 0.005
    movel([0.137159, -1.403046, -2.545607, -0.763736, 1.570796, 1.707955],accel_mss,speed_ms,0,blend_radius_m)
    speed_ms = 0.040
    # Splitting Linear movement in 2 (instruction 283: MoveL 262)
    movel([0.174820, -1.398287, -2.549118, -0.764984, 1.570796, 1.745617],accel_mss,speed_ms,0,blend_radius_m)
    movel([0.212258, -1.394754, -2.551703, -0.765932, 1.570796, 1.783055],accel_mss,speed_ms,0,blend_radius_m)
    speed_ms = 0.005
    movel([0.212258, -1.403290, -2.555604, -0.753495, 1.570796, 1.783055],accel_mss,speed_ms,0,blend_radius_m)
    speed_ms = 0.025
    movel([0.212995, -1.402513, -2.556178, -0.753699, 1.570796, 1.783791],accel_mss,speed_ms,0,blend_radius_m)
    movel([0.213276, -1.402201, -2.556407, -0.753780, 1.570796, 1.784073],accel_mss,speed_ms,0,blend_radius_m)
    movel([0.213298, -1.401947, -2.556595, -0.753847, 1.570796, 1.784095],accel_mss,speed_ms,0,blend_radius_m)
    movel([0.213229, -1.401814, -2.556693, -0.753882, 1.570796, 1.784026],accel_mss,speed_ms,0,blend_radius_m)
    movel([0.212929, -1.401746, -2.556743, -0.753900, 1.570796, 1.783725],accel_mss,speed_ms,0,blend_radius_m)
    movel([0.212539, -1.401942, -2.556598, -0.753848, 1.570796, 1.783336],accel_mss,speed_ms,0,blend_radius_m)
    movel([0.211824, -1.402619, -2.556099, -0.753671, 1.570796, 1.782621],accel_mss,speed_ms,0,blend_radius_m)
    movel([0.210769, -1.403737, -2.555273, -0.753378, 1.570796, 1.781565],accel_mss,speed_ms,0,blend_radius_m)
    movel([0.205843, -1.409184, -2.551224, -0.751981, 1.570796, 1.776640],accel_mss,speed_ms,0,blend_radius_m)
    movel([0.204956, -1.410043, -2.550582, -0.751764, 1.570796, 1.775752],accel_mss,speed_ms,0,blend_radius_m)
    movel([0.203263, -1.411446, -2.549530, -0.751413, 1.570796, 1.774059],accel_mss,speed_ms,0,blend_radius_m)
    movel([0.203180, -1.411391, -2.549571, -0.751427, 1.570796, 1.773976],accel_mss,speed_ms,0,blend_radius_m)
    movel([0.204405, -1.409407, -2.551058, -0.751924, 1.570796, 1.775201],accel_mss,speed_ms,0,blend_radius_m)
    movel([0.204693, -1.408783, -2.551524, -0.752082, 1.570796, 1.775490],accel_mss,speed_ms,0,blend_radius_m)
    movel([0.205056, -1.407571, -2.552428, -0.752390, 1.570796, 1.775853],accel_mss,speed_ms,0,blend_radius_m)
    movel([0.205078, -1.407327, -2.552610, -0.752452, 1.570796, 1.775875],accel_mss,speed_ms,0,blend_radius_m)
    movel([0.204845, -1.407180, -2.552720, -0.752490, 1.570796, 1.775641],accel_mss,speed_ms,0,blend_radius_m)
    movel([0.204649, -1.407237, -2.552677, -0.752475, 1.570796, 1.775445],accel_mss,speed_ms,0,blend_radius_m)
    movel([0.204084, -1.407646, -2.552372, -0.752371, 1.570796, 1.774880],accel_mss,speed_ms,0,blend_radius_m)
    movel([0.203703, -1.408009, -2.552101, -0.752278, 1.570796, 1.774499],accel_mss,speed_ms,0,blend_radius_m)
    movel([0.202377, -1.409088, -2.551296, -0.752005, 1.570796, 1.773173],accel_mss,speed_ms,0,blend_radius_m)
    movel([0.200783, -1.409954, -2.550648, -0.751787, 1.570796, 1.771579],accel_mss,speed_ms,0,blend_radius_m)
    movel([0.198815, -1.410647, -2.550129, -0.751613, 1.570796, 1.769612],accel_mss,speed_ms,0,blend_radius_m)
    movel([0.196342, -1.411216, -2.549702, -0.751470, 1.570796, 1.767138],accel_mss,speed_ms,0,blend_radius_m)
    movel([0.193574, -1.411606, -2.549409, -0.751373, 1.570796, 1.764370],accel_mss,speed_ms,0,blend_radius_m)
    movel([0.192481, -1.411670, -2.549362, -0.751357, 1.570796, 1.763278],accel_mss,speed_ms,0,blend_radius_m)
    movel([0.191968, -1.411589, -2.549422, -0.751377, 1.570796, 1.762764],accel_mss,speed_ms,0,blend_radius_m)
    movel([0.193125, -1.410815, -2.550003, -0.751571, 1.570796, 1.763921],accel_mss,speed_ms,0,blend_radius_m)
    movel([0.194094, -1.410188, -2.550473, -0.751728, 1.570796, 1.764890],accel_mss,speed_ms,0,blend_radius_m)
    movel([0.196326, -1.408364, -2.551836, -0.752188, 1.570796, 1.767122],accel_mss,speed_ms,0,blend_radius_m)
    movel([0.196574, -1.407967, -2.552133, -0.752289, 1.570796, 1.767371],accel_mss,speed_ms,0,blend_radius_m)
    movel([0.196504, -1.407757, -2.552290, -0.752343, 1.570796, 1.767301],accel_mss,speed_ms,0,blend_radius_m)
    movel([0.196205, -1.407640, -2.552376, -0.752372, 1.570796, 1.767001],accel_mss,speed_ms,0,blend_radius_m)
    movel([0.194383, -1.407610, -2.552399, -0.752380, 1.570796, 1.765179],accel_mss,speed_ms,0,blend_radius_m)
    movel([0.191988, -1.407594, -2.552411, -0.752384, 1.570796, 1.762784],accel_mss,speed_ms,0,blend_radius_m)
    movel([0.189879, -1.407394, -2.552560, -0.752435, 1.570796, 1.760675],accel_mss,speed_ms,0,blend_radius_m)
    movel([0.188178, -1.407036, -2.552827, -0.752527, 1.570796, 1.758974],accel_mss,speed_ms,0,blend_radius_m)
    movel([0.187061, -1.406523, -2.553208, -0.752658, 1.570796, 1.757858],accel_mss,speed_ms,0,blend_radius_m)
    movel([0.186560, -1.406179, -2.553464, -0.752746, 1.570796, 1.757356],accel_mss,speed_ms,0,blend_radius_m)
    movel([0.188628, -1.405758, -2.553777, -0.752855, 1.570796, 1.759424],accel_mss,speed_ms,0,blend_radius_m)
    movel([0.189090, -1.405630, -2.553872, -0.752888, 1.570796, 1.759886],accel_mss,speed_ms,0,blend_radius_m)
    movel([0.189607, -1.405360, -2.554072, -0.752957, 1.570796, 1.760404],accel_mss,speed_ms,0,blend_radius_m)
    movel([0.189781, -1.405074, -2.554284, -0.753031, 1.570796, 1.760578],accel_mss,speed_ms,0,blend_radius_m)
    movel([0.189749, -1.404838, -2.554459, -0.753092, 1.570796, 1.760546],accel_mss,speed_ms,0,blend_radius_m)
    movel([0.189456, -1.404622, -2.554619, -0.753148, 1.570796, 1.760252],accel_mss,speed_ms,0,blend_radius_m)
    movel([0.187133, -1.403654, -2.555335, -0.753400, 1.570796, 1.757929],accel_mss,speed_ms,0,blend_radius_m)
    movel([0.186609, -1.403384, -2.555534, -0.753470, 1.570796, 1.757405],accel_mss,speed_ms,0,blend_radius_m)
    movel([0.184440, -1.401938, -2.556601, -0.753850, 1.570796, 1.755236],accel_mss,speed_ms,0,blend_radius_m)
    movel([0.183283, -1.401048, -2.557256, -0.754084, 1.570796, 1.754079],accel_mss,speed_ms,0,blend_radius_m)
    movel([0.183316, -1.400879, -2.557381, -0.754129, 1.570796, 1.754112],accel_mss,speed_ms,0,blend_radius_m)
    movel([0.185288, -1.400773, -2.557459, -0.754157, 1.570796, 1.756084],accel_mss,speed_ms,0,blend_radius_m)
    movel([0.185716, -1.400735, -2.557486, -0.754167, 1.570796, 1.756513],accel_mss,speed_ms,0,blend_radius_m)
    movel([0.186580, -1.400524, -2.557642, -0.754223, 1.570796, 1.757376],accel_mss,speed_ms,0,blend_radius_m)
    movel([0.186686, -1.400404, -2.557730, -0.754255, 1.570796, 1.757482],accel_mss,speed_ms,0,blend_radius_m)
    movel([0.186743, -1.400027, -2.558007, -0.754355, 1.570796, 1.757539],accel_mss,speed_ms,0,blend_radius_m)
    movel([0.186632, -1.399840, -2.558143, -0.754405, 1.570796, 1.757428],accel_mss,speed_ms,0,blend_radius_m)
    movel([0.186087, -1.399438, -2.558439, -0.754512, 1.570796, 1.756883],accel_mss,speed_ms,0,blend_radius_m)
    movel([0.185288, -1.398908, -2.558827, -0.754654, 1.570796, 1.756085],accel_mss,speed_ms,0,blend_radius_m)
    movel([0.183948, -1.397503, -2.559855, -0.755032, 1.570796, 1.754744],accel_mss,speed_ms,0,blend_radius_m)
    movel([0.183403, -1.396649, -2.560478, -0.755263, 1.570796, 1.754199],accel_mss,speed_ms,0,blend_radius_m)
    movel([0.182615, -1.394728, -2.561875, -0.755786, 1.570796, 1.753411],accel_mss,speed_ms,0,blend_radius_m)
    movel([0.182409, -1.393739, -2.562593, -0.756058, 1.570796, 1.753206],accel_mss,speed_ms,0,blend_radius_m)
    movel([0.182291, -1.392006, -2.563846, -0.756537, 1.570796, 1.753087],accel_mss,speed_ms,0,blend_radius_m)
    movel([0.182169, -1.391624, -2.564122, -0.756643, 1.570796, 1.752965],accel_mss,speed_ms,0,blend_radius_m)
    movel([0.181958, -1.391488, -2.564220, -0.756681, 1.570796, 1.752755],accel_mss,speed_ms,0,blend_radius_m)
    movel([0.181659, -1.391545, -2.564179, -0.756665, 1.570796, 1.752455],accel_mss,speed_ms,0,blend_radius_m)
    movel([0.181400, -1.391841, -2.563966, -0.756583, 1.570796, 1.752196],accel_mss,speed_ms,0,blend_radius_m)
    movel([0.181291, -1.392472, -2.563509, -0.756407, 1.570796, 1.752087],accel_mss,speed_ms,0,blend_radius_m)
    movel([0.181467, -1.394567, -2.561992, -0.755830, 1.570796, 1.752263],accel_mss,speed_ms,0,blend_radius_m)
    movel([0.181772, -1.395809, -2.561089, -0.755491, 1.570796, 1.752569],accel_mss,speed_ms,0,blend_radius_m)
    movel([0.182255, -1.396984, -2.560233, -0.755172, 1.570796, 1.753052],accel_mss,speed_ms,0,blend_radius_m)
    movel([0.182893, -1.398044, -2.559459, -0.754886, 1.570796, 1.753689],accel_mss,speed_ms,0,blend_radius_m)
    movel([0.183660, -1.398936, -2.558807, -0.754647, 1.570796, 1.754457],accel_mss,speed_ms,0,blend_radius_m)
    movel([0.184310, -1.399597, -2.558322, -0.754470, 1.570796, 1.755106],accel_mss,speed_ms,0,blend_radius_m)
    movel([0.184284, -1.399801, -2.558173, -0.754416, 1.570796, 1.755080],accel_mss,speed_ms,0,blend_radius_m)
    movel([0.184058, -1.399908, -2.558094, -0.754387, 1.570796, 1.754854],accel_mss,speed_ms,0,blend_radius_m)
    movel([0.182268, -1.399637, -2.558293, -0.754459, 1.570796, 1.753064],accel_mss,speed_ms,0,blend_radius_m)
    movel([0.181785, -1.399641, -2.558290, -0.754458, 1.570796, 1.752582],accel_mss,speed_ms,0,blend_radius_m)
    movel([0.181463, -1.399746, -2.558213, -0.754430, 1.570796, 1.752259],accel_mss,speed_ms,0,blend_radius_m)
    movel([0.181244, -1.399951, -2.558063, -0.754376, 1.570796, 1.752041],accel_mss,speed_ms,0,blend_radius_m)
    movel([0.181142, -1.400289, -2.557814, -0.754286, 1.570796, 1.751939],accel_mss,speed_ms,0,blend_radius_m)
    movel([0.181245, -1.400557, -2.557618, -0.754215, 1.570796, 1.752041],accel_mss,speed_ms,0,blend_radius_m)
    movel([0.182830, -1.402051, -2.556518, -0.753820, 1.570796, 1.753626],accel_mss,speed_ms,0,blend_radius_m)
    movel([0.184632, -1.403489, -2.555457, -0.753443, 1.570796, 1.755428],accel_mss,speed_ms,0,blend_radius_m)
    movel([0.186344, -1.404506, -2.554705, -0.753178, 1.570796, 1.757140],accel_mss,speed_ms,0,blend_radius_m)
    movel([0.187606, -1.405119, -2.554250, -0.753020, 1.570796, 1.758402],accel_mss,speed_ms,0,blend_radius_m)
    movel([0.185027, -1.405403, -2.554040, -0.752946, 1.570796, 1.755823],accel_mss,speed_ms,0,blend_radius_m)
    movel([0.184789, -1.405518, -2.553955, -0.752917, 1.570796, 1.755586],accel_mss,speed_ms,0,blend_radius_m)
    movel([0.184643, -1.405700, -2.553819, -0.752870, 1.570796, 1.755439],accel_mss,speed_ms,0,blend_radius_m)
    movel([0.184621, -1.405981, -2.553611, -0.752797, 1.570796, 1.755417],accel_mss,speed_ms,0,blend_radius_m)
    movel([0.185170, -1.406657, -2.553109, -0.752624, 1.570796, 1.755967],accel_mss,speed_ms,0,blend_radius_m)
    movel([0.185790, -1.407106, -2.552774, -0.752509, 1.570796, 1.756586],accel_mss,speed_ms,0,blend_radius_m)
    movel([0.187086, -1.407758, -2.552289, -0.752342, 1.570796, 1.757882],accel_mss,speed_ms,0,blend_radius_m)
    movel([0.188753, -1.408215, -2.551948, -0.752226, 1.570796, 1.759550],accel_mss,speed_ms,0,blend_radius_m)
    movel([0.190790, -1.408477, -2.551752, -0.752160, 1.570796, 1.761587],accel_mss,speed_ms,0,blend_radius_m)
    movel([0.193192, -1.408549, -2.551699, -0.752141, 1.570796, 1.763988],accel_mss,speed_ms,0,blend_radius_m)
    movel([0.194924, -1.408578, -2.551677, -0.752134, 1.570796, 1.765720],accel_mss,speed_ms,0,blend_radius_m)
    movel([0.194195, -1.409218, -2.551199, -0.751972, 1.570796, 1.764991],accel_mss,speed_ms,0,blend_radius_m)
    movel([0.193477, -1.409740, -2.550808, -0.751840, 1.570796, 1.764273],accel_mss,speed_ms,0,blend_radius_m)
    movel([0.192591, -1.410271, -2.550411, -0.751707, 1.570796, 1.763387],accel_mss,speed_ms,0,blend_radius_m)
    movel([0.192107, -1.410480, -2.550254, -0.751654, 1.570796, 1.762903],accel_mss,speed_ms,0,blend_radius_m)
    movel([0.189930, -1.411314, -2.549629, -0.751446, 1.570796, 1.760726],accel_mss,speed_ms,0,blend_radius_m)
    movel([0.189718, -1.411474, -2.549509, -0.751406, 1.570796, 1.760514],accel_mss,speed_ms,0,blend_radius_m)
    movel([0.189584, -1.411841, -2.549233, -0.751315, 1.570796, 1.760380],accel_mss,speed_ms,0,blend_radius_m)
    movel([0.189686, -1.411980, -2.549128, -0.751280, 1.570796, 1.760482],accel_mss,speed_ms,0,blend_radius_m)
    movel([0.190443, -1.412256, -2.548921, -0.751212, 1.570796, 1.761239],accel_mss,speed_ms,0,blend_radius_m)
    movel([0.191620, -1.412496, -2.548741, -0.751152, 1.570796, 1.762416],accel_mss,speed_ms,0,blend_radius_m)
    movel([0.192758, -1.412563, -2.548690, -0.751136, 1.570796, 1.763554],accel_mss,speed_ms,0,blend_radius_m)
    movel([0.194091, -1.412458, -2.548769, -0.751162, 1.570796, 1.764887],accel_mss,speed_ms,0,blend_radius_m)
    movel([0.195886, -1.412169, -2.548987, -0.751233, 1.570796, 1.766682],accel_mss,speed_ms,0,blend_radius_m)
    movel([0.198116, -1.411680, -2.549354, -0.751355, 1.570796, 1.768912],accel_mss,speed_ms,0,blend_radius_m)
    movel([0.200023, -1.411101, -2.549789, -0.751499, 1.570796, 1.770820],accel_mss,speed_ms,0,blend_radius_m)
    movel([0.201628, -1.410430, -2.550292, -0.751667, 1.570796, 1.772424],accel_mss,speed_ms,0,blend_radius_m)
    movel([0.203338, -1.409405, -2.551059, -0.751925, 1.570796, 1.774134],accel_mss,speed_ms,0,blend_radius_m)
    movel([0.203201, -1.409950, -2.550651, -0.751788, 1.570796, 1.773997],accel_mss,speed_ms,0,blend_radius_m)
    movel([0.202513, -1.410874, -2.549959, -0.751556, 1.570796, 1.773309],accel_mss,speed_ms,0,blend_radius_m)
    movel([0.200977, -1.412626, -2.548643, -0.751120, 1.570796, 1.771773],accel_mss,speed_ms,0,blend_radius_m)
    movel([0.200127, -1.413545, -2.547951, -0.750893, 1.570796, 1.770923],accel_mss,speed_ms,0,blend_radius_m)
    movel([0.200034, -1.413754, -2.547793, -0.750842, 1.570796, 1.770830],accel_mss,speed_ms,0,blend_radius_m)
    movel([0.200107, -1.413914, -2.547672, -0.750803, 1.570796, 1.770903],accel_mss,speed_ms,0,blend_radius_m)
    movel([0.200330, -1.413971, -2.547629, -0.750788, 1.570796, 1.771126],accel_mss,speed_ms,0,blend_radius_m)
    movel([0.200605, -1.413902, -2.547682, -0.750806, 1.570796, 1.771401],accel_mss,speed_ms,0,blend_radius_m)
    movel([0.201876, -1.413238, -2.548182, -0.750969, 1.570796, 1.772672],accel_mss,speed_ms,0,blend_radius_m)
    movel([0.203545, -1.412158, -2.548995, -0.751236, 1.570796, 1.774341],accel_mss,speed_ms,0,blend_radius_m)
    movel([0.205114, -1.410881, -2.549954, -0.751554, 1.570796, 1.775911],accel_mss,speed_ms,0,blend_radius_m)
    movel([0.206889, -1.409139, -2.551258, -0.751992, 1.570796, 1.777686],accel_mss,speed_ms,0,blend_radius_m)
    movel([0.212258, -1.403290, -2.555604, -0.753495, 1.570796, 1.783055],accel_mss,speed_ms,0,blend_radius_m)
    movel([0.212995, -1.402513, -2.556178, -0.753699, 1.570796, 1.783791],accel_mss,speed_ms,0,blend_radius_m)
    movel([0.213276, -1.402201, -2.556407, -0.753780, 1.570796, 1.784073],accel_mss,speed_ms,0,blend_radius_m)
    movel([0.213298, -1.401947, -2.556595, -0.753847, 1.570796, 1.784095],accel_mss,speed_ms,0,blend_radius_m)
    movel([0.213229, -1.401814, -2.556693, -0.753882, 1.570796, 1.784026],accel_mss,speed_ms,0,blend_radius_m)
    movel([0.212929, -1.401746, -2.556743, -0.753900, 1.570796, 1.783725],accel_mss,speed_ms,0,blend_radius_m)
    movel([0.212699, -1.401863, -2.556657, -0.753869, 1.570796, 1.783495],accel_mss,speed_ms,0,blend_radius_m)
    speed_ms = 0.005
    movel([0.212699, -1.393317, -2.552749, -0.766323, 1.570796, 1.783495],accel_mss,speed_ms,0,blend_radius_m)
    speed_ms = 0.040
    movel([0.223035, -1.390420, -2.554849, -0.767120, 1.570796, 1.793831],accel_mss,speed_ms,0,blend_radius_m)
    speed_ms = 0.005
    movel([0.223035, -1.398987, -2.558769, -0.754633, 1.570796, 1.793831],accel_mss,speed_ms,0,blend_radius_m)
    speed_ms = 0.025
    movel([0.221622, -1.401960, -2.556585, -0.753844, 1.570796, 1.792419],accel_mss,speed_ms,0,blend_radius_m)
    movel([0.220878, -1.403325, -2.555578, -0.753486, 1.570796, 1.791674],accel_mss,speed_ms,0,blend_radius_m)
    movel([0.220530, -1.403722, -2.555285, -0.753382, 1.570796, 1.791326],accel_mss,speed_ms,0,blend_radius_m)
    movel([0.220197, -1.403883, -2.555166, -0.753340, 1.570796, 1.790993],accel_mss,speed_ms,0,blend_radius_m)
    movel([0.219990, -1.403812, -2.555218, -0.753359, 1.570796, 1.790786],accel_mss,speed_ms,0,blend_radius_m)
    movel([0.219920, -1.403447, -2.555488, -0.753454, 1.570796, 1.790716],accel_mss,speed_ms,0,blend_radius_m)
    movel([0.220087, -1.401791, -2.556710, -0.753888, 1.570796, 1.790883],accel_mss,speed_ms,0,blend_radius_m)
    movel([0.220082, -1.400837, -2.557411, -0.754140, 1.570796, 1.790878],accel_mss,speed_ms,0,blend_radius_m)
    movel([0.219829, -1.399377, -2.558483, -0.754529, 1.570796, 1.790626],accel_mss,speed_ms,0,blend_radius_m)
    movel([0.219704, -1.399196, -2.558616, -0.754577, 1.570796, 1.790500],accel_mss,speed_ms,0,blend_radius_m)
    movel([0.219580, -1.399230, -2.558591, -0.754568, 1.570796, 1.790377],accel_mss,speed_ms,0,blend_radius_m)
    movel([0.219406, -1.399501, -2.558393, -0.754496, 1.570796, 1.790202],accel_mss,speed_ms,0,blend_radius_m)
    movel([0.218116, -1.401972, -2.556576, -0.753841, 1.570796, 1.788912],accel_mss,speed_ms,0,blend_radius_m)
    movel([0.217283, -1.403349, -2.555560, -0.753480, 1.570796, 1.788080],accel_mss,speed_ms,0,blend_radius_m)
    movel([0.215067, -1.406593, -2.553156, -0.752640, 1.570796, 1.785863],accel_mss,speed_ms,0,blend_radius_m)
    movel([0.212805, -1.409599, -2.550914, -0.751876, 1.570796, 1.783601],accel_mss,speed_ms,0,blend_radius_m)
    movel([0.212393, -1.409968, -2.550638, -0.751783, 1.570796, 1.783189],accel_mss,speed_ms,0,blend_radius_m)
    movel([0.211898, -1.410161, -2.550493, -0.751734, 1.570796, 1.782695],accel_mss,speed_ms,0,blend_radius_m)
    movel([0.211633, -1.410150, -2.550502, -0.751737, 1.570796, 1.782429],accel_mss,speed_ms,0,blend_radius_m)
    movel([0.211528, -1.410014, -2.550603, -0.751772, 1.570796, 1.782325],accel_mss,speed_ms,0,blend_radius_m)
    movel([0.211850, -1.408859, -2.551467, -0.752063, 1.570796, 1.782646],accel_mss,speed_ms,0,blend_radius_m)
    movel([0.212004, -1.408385, -2.551821, -0.752183, 1.570796, 1.782801],accel_mss,speed_ms,0,blend_radius_m)
    movel([0.212282, -1.407186, -2.552715, -0.752488, 1.570796, 1.783079],accel_mss,speed_ms,0,blend_radius_m)
    movel([0.212315, -1.406648, -2.553115, -0.752626, 1.570796, 1.783112],accel_mss,speed_ms,0,blend_radius_m)
    movel([0.211063, -1.408506, -2.551730, -0.752152, 1.570796, 1.781860],accel_mss,speed_ms,0,blend_radius_m)
    movel([0.210390, -1.409336, -2.551111, -0.751942, 1.570796, 1.781186],accel_mss,speed_ms,0,blend_radius_m)
    movel([0.209789, -1.409958, -2.550646, -0.751786, 1.570796, 1.780585],accel_mss,speed_ms,0,blend_radius_m)
    movel([0.209427, -1.410149, -2.550502, -0.751738, 1.570796, 1.780223],accel_mss,speed_ms,0,blend_radius_m)
    movel([0.209173, -1.410089, -2.550547, -0.751753, 1.570796, 1.779969],accel_mss,speed_ms,0,blend_radius_m)
    movel([0.209149, -1.409854, -2.550723, -0.751812, 1.570796, 1.779945],accel_mss,speed_ms,0,blend_radius_m)
    movel([0.209438, -1.409325, -2.551119, -0.751945, 1.570796, 1.780234],accel_mss,speed_ms,0,blend_radius_m)
    movel([0.210196, -1.408261, -2.551914, -0.752214, 1.570796, 1.780992],accel_mss,speed_ms,0,blend_radius_m)
    movel([0.211644, -1.406034, -2.553572, -0.752784, 1.570796, 1.782440],accel_mss,speed_ms,0,blend_radius_m)
    movel([0.211950, -1.405460, -2.553998, -0.752932, 1.570796, 1.782747],accel_mss,speed_ms,0,blend_radius_m)
    movel([0.212654, -1.404233, -2.554907, -0.753249, 1.570796, 1.783450],accel_mss,speed_ms,0,blend_radius_m)
    movel([0.212908, -1.404069, -2.555028, -0.753292, 1.570796, 1.783704],accel_mss,speed_ms,0,blend_radius_m)
    movel([0.213185, -1.404069, -2.555028, -0.753292, 1.570796, 1.783982],accel_mss,speed_ms,0,blend_radius_m)
    movel([0.213379, -1.404302, -2.554856, -0.753231, 1.570796, 1.784175],accel_mss,speed_ms,0,blend_radius_m)
    movel([0.213443, -1.406098, -2.553524, -0.752767, 1.570796, 1.784240],accel_mss,speed_ms,0,blend_radius_m)
    movel([0.213317, -1.406936, -2.552901, -0.752552, 1.570796, 1.784113],accel_mss,speed_ms,0,blend_radius_m)
    movel([0.213218, -1.407521, -2.552466, -0.752403, 1.570796, 1.784014],accel_mss,speed_ms,0,blend_radius_m)
    movel([0.214514, -1.406075, -2.553541, -0.752773, 1.570796, 1.785310],accel_mss,speed_ms,0,blend_radius_m)
    movel([0.216040, -1.403732, -2.555277, -0.753380, 1.570796, 1.786837],accel_mss,speed_ms,0,blend_radius_m)
    movel([0.217555, -1.401188, -2.557153, -0.754047, 1.570796, 1.788351],accel_mss,speed_ms,0,blend_radius_m)
    movel([0.218670, -1.399031, -2.558737, -0.754621, 1.570796, 1.789467],accel_mss,speed_ms,0,blend_radius_m)
    movel([0.219430, -1.397599, -2.559784, -0.755006, 1.570796, 1.790226],accel_mss,speed_ms,0,blend_radius_m)
    movel([0.219682, -1.397400, -2.559930, -0.755059, 1.570796, 1.790478],accel_mss,speed_ms,0,blend_radius_m)
    movel([0.219963, -1.397354, -2.559963, -0.755072, 1.570796, 1.790759],accel_mss,speed_ms,0,blend_radius_m)
    movel([0.220247, -1.397546, -2.559823, -0.755020, 1.570796, 1.791044],accel_mss,speed_ms,0,blend_radius_m)
    movel([0.220910, -1.399062, -2.558714, -0.754613, 1.570796, 1.791706],accel_mss,speed_ms,0,blend_radius_m)
    movel([0.221105, -1.399905, -2.558096, -0.754388, 1.570796, 1.791902],accel_mss,speed_ms,0,blend_radius_m)
    movel([0.221255, -1.400846, -2.557405, -0.754138, 1.570796, 1.792051],accel_mss,speed_ms,0,blend_radius_m)
    movel([0.221709, -1.399953, -2.558061, -0.754375, 1.570796, 1.792505],accel_mss,speed_ms,0,blend_radius_m)
    movel([0.222279, -1.398413, -2.559189, -0.754787, 1.570796, 1.793075],accel_mss,speed_ms,0,blend_radius_m)
    movel([0.222646, -1.397154, -2.560109, -0.755126, 1.570796, 1.793443],accel_mss,speed_ms,0,blend_radius_m)
    movel([0.223915, -1.392529, -2.563468, -0.756391, 1.570796, 1.794711],accel_mss,speed_ms,0,blend_radius_m)
    movel([0.224136, -1.391932, -2.563899, -0.756557, 1.570796, 1.794932],accel_mss,speed_ms,0,blend_radius_m)
    movel([0.224329, -1.391719, -2.564054, -0.756617, 1.570796, 1.795125],accel_mss,speed_ms,0,blend_radius_m)
    movel([0.224575, -1.391644, -2.564108, -0.756637, 1.570796, 1.795371],accel_mss,speed_ms,0,blend_radius_m)
    movel([0.224750, -1.391722, -2.564052, -0.756616, 1.570796, 1.795546],accel_mss,speed_ms,0,blend_radius_m)
    movel([0.224833, -1.391979, -2.563866, -0.756544, 1.570796, 1.795629],accel_mss,speed_ms,0,blend_radius_m)
    movel([0.224581, -1.393716, -2.562609, -0.756064, 1.570796, 1.795378],accel_mss,speed_ms,0,blend_radius_m)
    movel([0.224081, -1.395688, -2.561177, -0.755524, 1.570796, 1.794877],accel_mss,speed_ms,0,blend_radius_m)
    movel([0.223511, -1.397665, -2.559736, -0.754988, 1.570796, 1.794307],accel_mss,speed_ms,0,blend_radius_m)
    movel([0.223034, -1.398989, -2.558767, -0.754632, 1.570796, 1.793831],accel_mss,speed_ms,0,blend_radius_m)
    movel([0.221985, -1.401194, -2.557149, -0.754046, 1.570796, 1.792782],accel_mss,speed_ms,0,blend_radius_m)
    speed_ms = 0.005
    movel([0.221985, -1.392643, -2.553239, -0.766507, 1.570796, 1.792782],accel_mss,speed_ms,0,blend_radius_m)
    speed_ms = 0.040
    movel([0.255061, -1.388949, -2.555911, -0.767529, 1.570796, 1.825858],accel_mss,speed_ms,0,blend_radius_m)
    speed_ms = 0.005
    movel([0.255061, -1.397526, -2.559838, -0.755025, 1.570796, 1.825858],accel_mss,speed_ms,0,blend_radius_m)
    speed_ms = 0.025
    movel([0.253552, -1.400586, -2.557596, -0.754207, 1.570796, 1.824348],accel_mss,speed_ms,0,blend_radius_m)
    movel([0.252674, -1.402160, -2.556438, -0.753791, 1.570796, 1.823471],accel_mss,speed_ms,0,blend_radius_m)
    movel([0.250934, -1.404950, -2.554376, -0.753063, 1.570796, 1.821731],accel_mss,speed_ms,0,blend_radius_m)
    movel([0.250464, -1.405581, -2.553908, -0.752900, 1.570796, 1.821261],accel_mss,speed_ms,0,blend_radius_m)
    movel([0.250118, -1.405893, -2.553676, -0.752820, 1.570796, 1.820915],accel_mss,speed_ms,0,blend_radius_m)
    movel([0.249786, -1.406008, -2.553591, -0.752790, 1.570796, 1.820583],accel_mss,speed_ms,0,blend_radius_m)
    movel([0.249527, -1.405863, -2.553698, -0.752827, 1.570796, 1.820323],accel_mss,speed_ms,0,blend_radius_m)
    movel([0.249527, -1.405643, -2.553861, -0.752884, 1.570796, 1.820323],accel_mss,speed_ms,0,blend_radius_m)
    movel([0.249972, -1.403100, -2.555744, -0.753545, 1.570796, 1.820768],accel_mss,speed_ms,0,blend_radius_m)
    movel([0.249142, -1.404436, -2.554757, -0.753197, 1.570796, 1.819939],accel_mss,speed_ms,0,blend_radius_m)
    movel([0.248264, -1.406008, -2.553591, -0.752790, 1.570796, 1.819061],accel_mss,speed_ms,0,blend_radius_m)
    movel([0.245914, -1.409646, -2.550879, -0.751864, 1.570796, 1.816711],accel_mss,speed_ms,0,blend_radius_m)
    movel([0.244439, -1.411718, -2.549326, -0.751345, 1.570796, 1.815235],accel_mss,speed_ms,0,blend_radius_m)
    movel([0.242292, -1.414551, -2.547192, -0.750647, 1.570796, 1.813088],accel_mss,speed_ms,0,blend_radius_m)
    movel([0.241911, -1.414865, -2.546954, -0.750570, 1.570796, 1.812708],accel_mss,speed_ms,0,blend_radius_m)
    movel([0.241609, -1.414902, -2.546926, -0.750561, 1.570796, 1.812405],accel_mss,speed_ms,0,blend_radius_m)
    movel([0.241510, -1.414810, -2.546996, -0.750583, 1.570796, 1.812306],accel_mss,speed_ms,0,blend_radius_m)
    movel([0.241487, -1.414463, -2.547258, -0.750668, 1.570796, 1.812283],accel_mss,speed_ms,0,blend_radius_m)
    movel([0.241563, -1.414182, -2.547470, -0.750737, 1.570796, 1.812359],accel_mss,speed_ms,0,blend_radius_m)
    movel([0.242015, -1.411980, -2.549128, -0.751280, 1.570796, 1.812812],accel_mss,speed_ms,0,blend_radius_m)
    movel([0.240170, -1.414423, -2.547288, -0.750678, 1.570796, 1.810966],accel_mss,speed_ms,0,blend_radius_m)
    movel([0.237663, -1.417569, -2.544905, -0.749915, 1.570796, 1.808459],accel_mss,speed_ms,0,blend_radius_m)
    movel([0.237041, -1.418284, -2.544361, -0.749744, 1.570796, 1.807837],accel_mss,speed_ms,0,blend_radius_m)
    movel([0.234233, -1.421186, -2.542147, -0.749056, 1.570796, 1.805030],accel_mss,speed_ms,0,blend_radius_m)
    movel([0.232819, -1.422555, -2.541097, -0.748736, 1.570796, 1.803615],accel_mss,speed_ms,0,blend_radius_m)
    movel([0.232506, -1.422717, -2.540974, -0.748699, 1.570796, 1.803303],accel_mss,speed_ms,0,blend_radius_m)
    movel([0.232261, -1.422680, -2.541002, -0.748707, 1.570796, 1.803057],accel_mss,speed_ms,0,blend_radius_m)
    movel([0.232133, -1.422509, -2.541133, -0.748747, 1.570796, 1.802930],accel_mss,speed_ms,0,blend_radius_m)
    movel([0.232153, -1.422219, -2.541355, -0.748815, 1.570796, 1.802950],accel_mss,speed_ms,0,blend_radius_m)
    movel([0.232681, -1.421239, -2.542106, -0.749044, 1.570796, 1.803477],accel_mss,speed_ms,0,blend_radius_m)
    movel([0.232611, -1.421180, -2.542151, -0.749058, 1.570796, 1.803408],accel_mss,speed_ms,0,blend_radius_m)
    movel([0.232354, -1.421366, -2.542009, -0.749014, 1.570796, 1.803151],accel_mss,speed_ms,0,blend_radius_m)
    movel([0.231596, -1.422195, -2.541374, -0.748820, 1.570796, 1.802392],accel_mss,speed_ms,0,blend_radius_m)
    movel([0.230421, -1.423426, -2.540429, -0.748534, 1.570796, 1.801217],accel_mss,speed_ms,0,blend_radius_m)
    movel([0.229169, -1.424600, -2.539525, -0.748264, 1.570796, 1.799966],accel_mss,speed_ms,0,blend_radius_m)
    movel([0.226205, -1.427040, -2.537641, -0.747708, 1.570796, 1.797001],accel_mss,speed_ms,0,blend_radius_m)
    movel([0.222819, -1.429428, -2.535788, -0.747173, 1.570796, 1.793616],accel_mss,speed_ms,0,blend_radius_m)
    movel([0.218255, -1.432172, -2.533648, -0.746569, 1.570796, 1.789051],accel_mss,speed_ms,0,blend_radius_m)
    movel([0.217773, -1.432408, -2.533464, -0.746517, 1.570796, 1.788569],accel_mss,speed_ms,0,blend_radius_m)
    movel([0.217478, -1.432500, -2.533392, -0.746497, 1.570796, 1.788274],accel_mss,speed_ms,0,blend_radius_m)
    movel([0.217301, -1.432470, -2.533415, -0.746504, 1.570796, 1.788097],accel_mss,speed_ms,0,blend_radius_m)
    movel([0.217147, -1.432138, -2.533675, -0.746576, 1.570796, 1.787944],accel_mss,speed_ms,0,blend_radius_m)
    movel([0.217236, -1.432021, -2.533766, -0.746602, 1.570796, 1.788033],accel_mss,speed_ms,0,blend_radius_m)
    movel([0.219260, -1.430742, -2.534765, -0.746882, 1.570796, 1.790056],accel_mss,speed_ms,0,blend_radius_m)
    movel([0.221369, -1.429468, -2.535757, -0.747164, 1.570796, 1.792165],accel_mss,speed_ms,0,blend_radius_m)
    movel([0.223451, -1.428126, -2.536799, -0.747464, 1.570796, 1.794247],accel_mss,speed_ms,0,blend_radius_m)
    movel([0.225214, -1.426889, -2.537758, -0.747742, 1.570796, 1.796011],accel_mss,speed_ms,0,blend_radius_m)
    movel([0.226922, -1.425572, -2.538775, -0.748041, 1.570796, 1.797718],accel_mss,speed_ms,0,blend_radius_m)
    movel([0.228407, -1.424302, -2.539755, -0.748332, 1.570796, 1.799203],accel_mss,speed_ms,0,blend_radius_m)
    movel([0.229817, -1.422963, -2.540784, -0.748642, 1.570796, 1.800613],accel_mss,speed_ms,0,blend_radius_m)
    movel([0.231095, -1.421602, -2.541828, -0.748959, 1.570796, 1.801891],accel_mss,speed_ms,0,blend_radius_m)
    movel([0.233309, -1.418941, -2.543861, -0.749587, 1.570796, 1.804105],accel_mss,speed_ms,0,blend_radius_m)
    movel([0.233578, -1.418718, -2.544031, -0.749640, 1.570796, 1.804374],accel_mss,speed_ms,0,blend_radius_m)
    movel([0.233888, -1.418589, -2.544129, -0.749671, 1.570796, 1.804685],accel_mss,speed_ms,0,blend_radius_m)
    movel([0.234100, -1.418612, -2.544111, -0.749665, 1.570796, 1.804896],accel_mss,speed_ms,0,blend_radius_m)
    movel([0.234173, -1.418778, -2.543985, -0.749626, 1.570796, 1.804969],accel_mss,speed_ms,0,blend_radius_m)
    movel([0.234003, -1.419782, -2.543219, -0.749387, 1.570796, 1.804799],accel_mss,speed_ms,0,blend_radius_m)
    movel([0.233940, -1.420303, -2.542822, -0.749264, 1.570796, 1.804736],accel_mss,speed_ms,0,blend_radius_m)
    movel([0.234406, -1.419954, -2.543088, -0.749347, 1.570796, 1.805202],accel_mss,speed_ms,0,blend_radius_m)
    movel([0.234802, -1.419557, -2.543391, -0.749441, 1.570796, 1.805599],accel_mss,speed_ms,0,blend_radius_m)
    movel([0.236870, -1.417305, -2.545105, -0.749978, 1.570796, 1.807667],accel_mss,speed_ms,0,blend_radius_m)
    movel([0.238322, -1.415577, -2.546416, -0.750396, 1.570796, 1.809118],accel_mss,speed_ms,0,blend_radius_m)
    movel([0.239682, -1.413808, -2.547752, -0.750829, 1.570796, 1.810478],accel_mss,speed_ms,0,blend_radius_m)
    movel([0.241023, -1.411908, -2.549183, -0.751298, 1.570796, 1.811819],accel_mss,speed_ms,0,blend_radius_m)
    movel([0.242135, -1.410381, -2.550329, -0.751679, 1.570796, 1.812931],accel_mss,speed_ms,0,blend_radius_m)
    movel([0.242308, -1.410203, -2.550462, -0.751724, 1.570796, 1.813104],accel_mss,speed_ms,0,blend_radius_m)
    movel([0.242602, -1.410029, -2.550592, -0.751768, 1.570796, 1.813398],accel_mss,speed_ms,0,blend_radius_m)
    movel([0.242697, -1.410069, -2.550562, -0.751758, 1.570796, 1.813494],accel_mss,speed_ms,0,blend_radius_m)
    movel([0.242907, -1.410397, -2.550316, -0.751675, 1.570796, 1.813703],accel_mss,speed_ms,0,blend_radius_m)
    movel([0.242964, -1.410702, -2.550088, -0.751599, 1.570796, 1.813760],accel_mss,speed_ms,0,blend_radius_m)
    movel([0.242962, -1.412354, -2.548847, -0.751187, 1.570796, 1.813758],accel_mss,speed_ms,0,blend_radius_m)
    movel([0.243680, -1.411419, -2.549550, -0.751420, 1.570796, 1.814476],accel_mss,speed_ms,0,blend_radius_m)
    movel([0.245231, -1.409281, -2.551152, -0.751956, 1.570796, 1.816028],accel_mss,speed_ms,0,blend_radius_m)
    movel([0.246721, -1.406990, -2.552861, -0.752538, 1.570796, 1.817517],accel_mss,speed_ms,0,blend_radius_m)
    movel([0.247996, -1.404795, -2.554490, -0.753103, 1.570796, 1.818792],accel_mss,speed_ms,0,blend_radius_m)
    movel([0.248884, -1.402964, -2.555845, -0.753580, 1.570796, 1.819681],accel_mss,speed_ms,0,blend_radius_m)
    movel([0.249660, -1.401257, -2.557103, -0.754029, 1.570796, 1.820457],accel_mss,speed_ms,0,blend_radius_m)
    movel([0.249866, -1.401033, -2.557267, -0.754088, 1.570796, 1.820663],accel_mss,speed_ms,0,blend_radius_m)
    movel([0.250116, -1.400925, -2.557347, -0.754117, 1.570796, 1.820912],accel_mss,speed_ms,0,blend_radius_m)
    movel([0.250385, -1.400977, -2.557309, -0.754103, 1.570796, 1.821181],accel_mss,speed_ms,0,blend_radius_m)
    movel([0.250773, -1.401670, -2.556799, -0.753920, 1.570796, 1.821569],accel_mss,speed_ms,0,blend_radius_m)
    movel([0.250930, -1.402398, -2.556263, -0.753729, 1.570796, 1.821726],accel_mss,speed_ms,0,blend_radius_m)
    movel([0.251075, -1.403222, -2.555654, -0.753513, 1.570796, 1.821871],accel_mss,speed_ms,0,blend_radius_m)
    movel([0.251862, -1.401901, -2.556628, -0.753859, 1.570796, 1.822659],accel_mss,speed_ms,0,blend_radius_m)
    movel([0.253507, -1.398819, -2.558892, -0.754678, 1.570796, 1.824303],accel_mss,speed_ms,0,blend_radius_m)
    movel([0.254273, -1.397131, -2.560126, -0.755132, 1.570796, 1.825069],accel_mss,speed_ms,0,blend_radius_m)
    movel([0.255673, -1.393717, -2.562609, -0.756064, 1.570796, 1.826469],accel_mss,speed_ms,0,blend_radius_m)
    movel([0.255878, -1.393390, -2.562846, -0.756154, 1.570796, 1.826675],accel_mss,speed_ms,0,blend_radius_m)
    movel([0.256084, -1.393232, -2.562960, -0.756197, 1.570796, 1.826881],accel_mss,speed_ms,0,blend_radius_m)
    movel([0.256444, -1.393164, -2.563009, -0.756216, 1.570796, 1.827240],accel_mss,speed_ms,0,blend_radius_m)
    movel([0.256599, -1.393299, -2.562911, -0.756179, 1.570796, 1.827395],accel_mss,speed_ms,0,blend_radius_m)
    movel([0.256551, -1.393708, -2.562615, -0.756066, 1.570796, 1.827348],accel_mss,speed_ms,0,blend_radius_m)
    movel([0.255355, -1.396845, -2.560335, -0.755209, 1.570796, 1.826152],accel_mss,speed_ms,0,blend_radius_m)
    movel([0.255061, -1.397526, -2.559838, -0.755025, 1.570796, 1.825858],accel_mss,speed_ms,0,blend_radius_m)
    movel([0.253971, -1.399734, -2.558222, -0.754433, 1.570796, 1.824767],accel_mss,speed_ms,0,blend_radius_m)
    speed_ms = 0.005
    movel([0.253971, -1.391173, -2.554305, -0.766912, 1.570796, 1.824767],accel_mss,speed_ms,0,blend_radius_m)
    speed_ms = 0.040
    movel([0.291751, -1.365864, -2.572169, -0.774356, 1.570796, 1.862547],accel_mss,speed_ms,0,blend_radius_m)
    speed_ms = 0.005
    movel([0.291751, -1.374603, -2.576196, -0.761590, 1.570796, 1.862547],accel_mss,speed_ms,0,blend_radius_m)
    speed_ms = 0.025
    movel([0.289793, -1.378338, -2.573582, -0.760469, 1.570796, 1.860589],accel_mss,speed_ms,0,blend_radius_m)
    movel([0.287266, -1.382450, -2.570681, -0.759258, 1.570796, 1.858062],accel_mss,speed_ms,0,blend_radius_m)
    movel([0.284520, -1.386421, -2.567857, -0.758111, 1.570796, 1.855316],accel_mss,speed_ms,0,blend_radius_m)
    movel([0.283243, -1.388094, -2.566661, -0.757635, 1.570796, 1.854039],accel_mss,speed_ms,0,blend_radius_m)
    movel([0.280417, -1.391356, -2.564315, -0.756717, 1.570796, 1.851213],accel_mss,speed_ms,0,blend_radius_m)
    movel([0.278866, -1.392927, -2.563180, -0.756281, 1.570796, 1.849663],accel_mss,speed_ms,0,blend_radius_m)
    movel([0.277250, -1.394427, -2.562094, -0.755868, 1.570796, 1.848046],accel_mss,speed_ms,0,blend_radius_m)
    movel([0.275565, -1.395856, -2.561055, -0.755478, 1.570796, 1.846361],accel_mss,speed_ms,0,blend_radius_m)
    movel([0.273908, -1.397139, -2.560120, -0.755130, 1.570796, 1.844704],accel_mss,speed_ms,0,blend_radius_m)
    movel([0.272199, -1.398341, -2.559242, -0.754806, 1.570796, 1.842995],accel_mss,speed_ms,0,blend_radius_m)
    movel([0.270616, -1.399330, -2.558518, -0.754541, 1.570796, 1.841412],accel_mss,speed_ms,0,blend_radius_m)
    movel([0.268994, -1.400203, -2.557878, -0.754309, 1.570796, 1.839790],accel_mss,speed_ms,0,blend_radius_m)
    movel([0.267616, -1.400835, -2.557413, -0.754141, 1.570796, 1.838412],accel_mss,speed_ms,0,blend_radius_m)
    movel([0.266449, -1.401260, -2.557100, -0.754028, 1.570796, 1.837245],accel_mss,speed_ms,0,blend_radius_m)
    movel([0.265318, -1.401535, -2.556898, -0.753956, 1.570796, 1.836114],accel_mss,speed_ms,0,blend_radius_m)
    movel([0.264065, -1.401705, -2.556773, -0.753911, 1.570796, 1.834862],accel_mss,speed_ms,0,blend_radius_m)
    movel([0.262836, -1.401720, -2.556762, -0.753907, 1.570796, 1.833632],accel_mss,speed_ms,0,blend_radius_m)
    movel([0.261779, -1.401531, -2.556901, -0.753957, 1.570796, 1.832576],accel_mss,speed_ms,0,blend_radius_m)
    movel([0.260848, -1.401121, -2.557203, -0.754065, 1.570796, 1.831644],accel_mss,speed_ms,0,blend_radius_m)
    movel([0.259995, -1.400475, -2.557677, -0.754236, 1.570796, 1.830791],accel_mss,speed_ms,0,blend_radius_m)
    movel([0.259086, -1.399346, -2.558506, -0.754537, 1.570796, 1.829882],accel_mss,speed_ms,0,blend_radius_m)
    movel([0.258408, -1.397871, -2.559585, -0.754932, 1.570796, 1.829205],accel_mss,speed_ms,0,blend_radius_m)
    movel([0.257879, -1.395851, -2.561059, -0.755479, 1.570796, 1.828676],accel_mss,speed_ms,0,blend_radius_m)
    movel([0.257435, -1.392981, -2.563141, -0.756266, 1.570796, 1.828231],accel_mss,speed_ms,0,blend_radius_m)
    movel([0.257015, -1.390281, -2.565090, -0.757018, 1.570796, 1.827811],accel_mss,speed_ms,0,blend_radius_m)
    movel([0.256803, -1.389621, -2.565564, -0.757203, 1.570796, 1.827600],accel_mss,speed_ms,0,blend_radius_m)
    movel([0.256224, -1.388669, -2.566249, -0.757472, 1.570796, 1.827020],accel_mss,speed_ms,0,blend_radius_m)
    movel([0.255974, -1.389160, -2.565896, -0.757333, 1.570796, 1.826770],accel_mss,speed_ms,0,blend_radius_m)
    movel([0.255184, -1.390576, -2.564877, -0.756935, 1.570796, 1.825980],accel_mss,speed_ms,0,blend_radius_m)
    movel([0.254281, -1.391965, -2.563876, -0.756548, 1.570796, 1.825077],accel_mss,speed_ms,0,blend_radius_m)
    movel([0.250614, -1.397092, -2.560155, -0.755143, 1.570796, 1.821410],accel_mss,speed_ms,0,blend_radius_m)
    movel([0.246685, -1.402324, -2.556317, -0.753748, 1.570796, 1.817482],accel_mss,speed_ms,0,blend_radius_m)
    movel([0.243531, -1.406182, -2.553461, -0.752745, 1.570796, 1.814327],accel_mss,speed_ms,0,blend_radius_m)
    movel([0.239923, -1.410131, -2.550516, -0.751742, 1.570796, 1.810719],accel_mss,speed_ms,0,blend_radius_m)
    movel([0.234712, -1.415431, -2.546526, -0.750432, 1.570796, 1.805508],accel_mss,speed_ms,0,blend_radius_m)
    movel([0.229342, -1.420688, -2.542528, -0.749173, 1.570796, 1.800139],accel_mss,speed_ms,0,blend_radius_m)
    movel([0.225081, -1.424606, -2.539521, -0.748262, 1.570796, 1.795877],accel_mss,speed_ms,0,blend_radius_m)
    movel([0.222345, -1.426874, -2.537769, -0.747746, 1.570796, 1.793141],accel_mss,speed_ms,0,blend_radius_m)
    movel([0.219496, -1.428960, -2.536152, -0.747277, 1.570796, 1.790292],accel_mss,speed_ms,0,blend_radius_m)
    movel([0.216974, -1.430596, -2.534879, -0.746914, 1.570796, 1.787771],accel_mss,speed_ms,0,blend_radius_m)
    movel([0.216382, -1.430870, -2.534665, -0.746854, 1.570796, 1.787179],accel_mss,speed_ms,0,blend_radius_m)
    movel([0.215794, -1.430979, -2.534580, -0.746830, 1.570796, 1.786590],accel_mss,speed_ms,0,blend_radius_m)
    movel([0.215617, -1.430912, -2.534632, -0.746845, 1.570796, 1.786413],accel_mss,speed_ms,0,blend_radius_m)
    movel([0.215565, -1.430725, -2.534778, -0.746886, 1.570796, 1.786361],accel_mss,speed_ms,0,blend_radius_m)
    movel([0.216415, -1.427307, -2.537434, -0.747648, 1.570796, 1.787211],accel_mss,speed_ms,0,blend_radius_m)
    movel([0.216420, -1.427022, -2.537655, -0.747712, 1.570796, 1.787216],accel_mss,speed_ms,0,blend_radius_m)
    movel([0.216306, -1.426794, -2.537831, -0.747764, 1.570796, 1.787103],accel_mss,speed_ms,0,blend_radius_m)
    movel([0.216097, -1.426689, -2.537912, -0.747787, 1.570796, 1.786894],accel_mss,speed_ms,0,blend_radius_m)
    movel([0.215812, -1.426717, -2.537891, -0.747781, 1.570796, 1.786608],accel_mss,speed_ms,0,blend_radius_m)
    movel([0.214397, -1.427239, -2.537487, -0.747663, 1.570796, 1.785193],accel_mss,speed_ms,0,blend_radius_m)
    movel([0.213045, -1.427689, -2.537138, -0.747562, 1.570796, 1.783841],accel_mss,speed_ms,0,blend_radius_m)
    movel([0.211654, -1.427944, -2.536941, -0.747505, 1.570796, 1.782450],accel_mss,speed_ms,0,blend_radius_m)
    movel([0.210504, -1.427975, -2.536917, -0.747498, 1.570796, 1.781300],accel_mss,speed_ms,0,blend_radius_m)
    movel([0.210198, -1.427899, -2.536975, -0.747515, 1.570796, 1.780995],accel_mss,speed_ms,0,blend_radius_m)
    movel([0.209935, -1.427589, -2.537216, -0.747584, 1.570796, 1.780731],accel_mss,speed_ms,0,blend_radius_m)
    movel([0.209927, -1.427417, -2.537349, -0.747623, 1.570796, 1.780723],accel_mss,speed_ms,0,blend_radius_m)
    movel([0.210132, -1.426593, -2.537987, -0.747809, 1.570796, 1.780929],accel_mss,speed_ms,0,blend_radius_m)
    movel([0.210084, -1.426449, -2.538098, -0.747842, 1.570796, 1.780880],accel_mss,speed_ms,0,blend_radius_m)
    movel([0.209719, -1.426244, -2.538257, -0.747888, 1.570796, 1.780515],accel_mss,speed_ms,0,blend_radius_m)
    movel([0.209366, -1.426308, -2.538207, -0.747874, 1.570796, 1.780162],accel_mss,speed_ms,0,blend_radius_m)
    movel([0.204990, -1.428219, -2.536727, -0.747443, 1.570796, 1.775787],accel_mss,speed_ms,0,blend_radius_m)
    movel([0.204206, -1.428539, -2.536479, -0.747371, 1.570796, 1.775002],accel_mss,speed_ms,0,blend_radius_m)
    movel([0.203982, -1.428523, -2.536491, -0.747375, 1.570796, 1.774778],accel_mss,speed_ms,0,blend_radius_m)
    movel([0.203936, -1.428442, -2.536555, -0.747393, 1.570796, 1.774733],accel_mss,speed_ms,0,blend_radius_m)
    movel([0.203933, -1.428205, -2.536738, -0.747446, 1.570796, 1.774729],accel_mss,speed_ms,0,blend_radius_m)
    movel([0.204029, -1.428021, -2.536881, -0.747487, 1.570796, 1.774825],accel_mss,speed_ms,0,blend_radius_m)
    movel([0.204562, -1.427574, -2.537227, -0.747588, 1.570796, 1.775358],accel_mss,speed_ms,0,blend_radius_m)
    movel([0.205072, -1.427256, -2.537474, -0.747659, 1.570796, 1.775868],accel_mss,speed_ms,0,blend_radius_m)
    movel([0.207229, -1.425859, -2.538554, -0.747976, 1.570796, 1.778025],accel_mss,speed_ms,0,blend_radius_m)
    movel([0.209281, -1.424292, -2.539763, -0.748335, 1.570796, 1.780077],accel_mss,speed_ms,0,blend_radius_m)
    movel([0.211751, -1.422167, -2.541395, -0.748827, 1.570796, 1.782547],accel_mss,speed_ms,0,blend_radius_m)
    movel([0.214131, -1.419949, -2.543092, -0.749348, 1.570796, 1.784927],accel_mss,speed_ms,0,blend_radius_m)
    movel([0.216600, -1.417467, -2.544982, -0.749940, 1.570796, 1.787397],accel_mss,speed_ms,0,blend_radius_m)
    movel([0.218963, -1.414903, -2.546925, -0.750560, 1.570796, 1.789759],accel_mss,speed_ms,0,blend_radius_m)
    movel([0.221111, -1.412367, -2.548838, -0.751184, 1.570796, 1.791907],accel_mss,speed_ms,0,blend_radius_m)
    movel([0.223124, -1.409760, -2.550794, -0.751835, 1.570796, 1.793921],accel_mss,speed_ms,0,blend_radius_m)
    movel([0.224374, -1.407947, -2.552148, -0.752294, 1.570796, 1.795171],accel_mss,speed_ms,0,blend_radius_m)
    movel([0.225478, -1.406095, -2.553526, -0.752768, 1.570796, 1.796275],accel_mss,speed_ms,0,blend_radius_m)
    movel([0.226323, -1.404386, -2.554793, -0.753209, 1.570796, 1.797119],accel_mss,speed_ms,0,blend_radius_m)
    movel([0.226966, -1.402675, -2.556058, -0.753656, 1.570796, 1.797763],accel_mss,speed_ms,0,blend_radius_m)
    movel([0.227410, -1.400952, -2.557327, -0.754110, 1.570796, 1.798206],accel_mss,speed_ms,0,blend_radius_m)
    movel([0.227643, -1.399267, -2.558564, -0.754558, 1.570796, 1.798439],accel_mss,speed_ms,0,blend_radius_m)
    movel([0.227697, -1.397423, -2.559912, -0.755053, 1.570796, 1.798493],accel_mss,speed_ms,0,blend_radius_m)
    movel([0.227579, -1.395637, -2.561215, -0.755538, 1.570796, 1.798375],accel_mss,speed_ms,0,blend_radius_m)
    movel([0.227326, -1.394200, -2.562258, -0.755931, 1.570796, 1.798123],accel_mss,speed_ms,0,blend_radius_m)
    movel([0.226871, -1.392562, -2.563444, -0.756382, 1.570796, 1.797667],accel_mss,speed_ms,0,blend_radius_m)
    movel([0.226339, -1.391082, -2.564513, -0.756794, 1.570796, 1.797135],accel_mss,speed_ms,0,blend_radius_m)
    movel([0.225869, -1.390290, -2.565084, -0.757016, 1.570796, 1.796665],accel_mss,speed_ms,0,blend_radius_m)
    movel([0.225194, -1.389726, -2.565489, -0.757174, 1.570796, 1.795990],accel_mss,speed_ms,0,blend_radius_m)
    movel([0.224364, -1.389463, -2.565678, -0.757248, 1.570796, 1.795160],accel_mss,speed_ms,0,blend_radius_m)
    movel([0.223374, -1.389509, -2.565645, -0.757235, 1.570796, 1.794171],accel_mss,speed_ms,0,blend_radius_m)
    movel([0.222237, -1.389858, -2.565395, -0.757137, 1.570796, 1.793034],accel_mss,speed_ms,0,blend_radius_m)
    movel([0.221463, -1.390284, -2.565088, -0.757017, 1.570796, 1.792259],accel_mss,speed_ms,0,blend_radius_m)
    movel([0.220675, -1.390914, -2.564634, -0.756841, 1.570796, 1.791471],accel_mss,speed_ms,0,blend_radius_m)
    movel([0.219803, -1.391818, -2.563982, -0.756589, 1.570796, 1.790599],accel_mss,speed_ms,0,blend_radius_m)
    movel([0.218750, -1.393101, -2.563055, -0.756233, 1.570796, 1.789547],accel_mss,speed_ms,0,blend_radius_m)
    movel([0.216024, -1.396322, -2.560716, -0.755351, 1.570796, 1.786820],accel_mss,speed_ms,0,blend_radius_m)
    movel([0.214669, -1.397736, -2.559684, -0.754969, 1.570796, 1.785465],accel_mss,speed_ms,0,blend_radius_m)
    movel([0.213239, -1.399090, -2.558693, -0.754605, 1.570796, 1.784035],accel_mss,speed_ms,0,blend_radius_m)
    movel([0.211880, -1.400257, -2.557838, -0.754294, 1.570796, 1.782677],accel_mss,speed_ms,0,blend_radius_m)
    movel([0.210461, -1.401350, -2.557034, -0.754005, 1.570796, 1.781258],accel_mss,speed_ms,0,blend_radius_m)
    movel([0.209140, -1.402246, -2.556375, -0.753769, 1.570796, 1.779936],accel_mss,speed_ms,0,blend_radius_m)
    movel([0.207772, -1.403032, -2.555795, -0.753563, 1.570796, 1.778569],accel_mss,speed_ms,0,blend_radius_m)
    movel([0.205590, -1.404005, -2.555075, -0.753309, 1.570796, 1.776386],accel_mss,speed_ms,0,blend_radius_m)
    movel([0.203405, -1.404635, -2.554609, -0.753145, 1.570796, 1.774202],accel_mss,speed_ms,0,blend_radius_m)
    movel([0.201172, -1.404945, -2.554380, -0.753065, 1.570796, 1.771968],accel_mss,speed_ms,0,blend_radius_m)
    movel([0.199062, -1.404921, -2.554397, -0.753071, 1.570796, 1.769858],accel_mss,speed_ms,0,blend_radius_m)
    movel([0.196999, -1.404549, -2.554673, -0.753167, 1.570796, 1.767795],accel_mss,speed_ms,0,blend_radius_m)
    movel([0.195155, -1.403858, -2.555184, -0.753347, 1.570796, 1.765952],accel_mss,speed_ms,0,blend_radius_m)
    movel([0.193479, -1.402829, -2.555944, -0.753616, 1.570796, 1.764275],accel_mss,speed_ms,0,blend_radius_m)
    movel([0.192069, -1.401537, -2.556897, -0.753955, 1.570796, 1.762865],accel_mss,speed_ms,0,blend_radius_m)
    movel([0.191110, -1.400341, -2.557776, -0.754272, 1.570796, 1.761906],accel_mss,speed_ms,0,blend_radius_m)
    movel([0.190279, -1.399047, -2.558725, -0.754617, 1.570796, 1.761075],accel_mss,speed_ms,0,blend_radius_m)
    movel([0.189442, -1.397458, -2.559887, -0.755044, 1.570796, 1.760238],accel_mss,speed_ms,0,blend_radius_m)
    movel([0.188032, -1.393972, -2.562424, -0.755993, 1.570796, 1.758829],accel_mss,speed_ms,0,blend_radius_m)
    movel([0.187465, -1.392079, -2.563794, -0.756516, 1.570796, 1.758261],accel_mss,speed_ms,0,blend_radius_m)
    movel([0.186665, -1.388149, -2.566621, -0.757619, 1.570796, 1.757462],accel_mss,speed_ms,0,blend_radius_m)
    movel([0.186398, -1.385484, -2.568526, -0.758379, 1.570796, 1.757194],accel_mss,speed_ms,0,blend_radius_m)
    movel([0.186334, -1.382729, -2.570483, -0.759176, 1.570796, 1.757131],accel_mss,speed_ms,0,blend_radius_m)
    movel([0.186490, -1.380002, -2.572411, -0.759976, 1.570796, 1.757286],accel_mss,speed_ms,0,blend_radius_m)
    movel([0.186871, -1.377199, -2.574381, -0.760809, 1.570796, 1.757667],accel_mss,speed_ms,0,blend_radius_m)
    movel([0.187456, -1.374488, -2.576276, -0.761625, 1.570796, 1.758252],accel_mss,speed_ms,0,blend_radius_m)
    movel([0.188266, -1.371728, -2.578194, -0.762467, 1.570796, 1.759062],accel_mss,speed_ms,0,blend_radius_m)
    movel([0.189256, -1.369119, -2.579997, -0.763273, 1.570796, 1.760052],accel_mss,speed_ms,0,blend_radius_m)
    movel([0.190498, -1.366496, -2.581801, -0.764093, 1.570796, 1.761294],accel_mss,speed_ms,0,blend_radius_m)
    movel([0.191485, -1.364781, -2.582974, -0.764634, 1.570796, 1.762281],accel_mss,speed_ms,0,blend_radius_m)
    movel([0.192852, -1.362721, -2.584378, -0.765290, 1.570796, 1.763648],accel_mss,speed_ms,0,blend_radius_m)
    movel([0.194334, -1.360695, -2.585754, -0.765940, 1.570796, 1.765131],accel_mss,speed_ms,0,blend_radius_m)
    movel([0.195665, -1.359088, -2.586841, -0.766461, 1.570796, 1.766461],accel_mss,speed_ms,0,blend_radius_m)
    movel([0.197068, -1.357605, -2.587840, -0.766944, 1.570796, 1.767864],accel_mss,speed_ms,0,blend_radius_m)
    movel([0.200218, -1.354712, -2.589781, -0.767895, 1.570796, 1.771015],accel_mss,speed_ms,0,blend_radius_m)
    movel([0.201132, -1.354088, -2.590199, -0.768102, 1.570796, 1.771928],accel_mss,speed_ms,0,blend_radius_m)
    movel([0.201841, -1.353771, -2.590411, -0.768207, 1.570796, 1.772637],accel_mss,speed_ms,0,blend_radius_m)
    movel([0.202545, -1.353588, -2.590533, -0.768268, 1.570796, 1.773341],accel_mss,speed_ms,0,blend_radius_m)
    movel([0.203189, -1.353553, -2.590556, -0.768280, 1.570796, 1.773985],accel_mss,speed_ms,0,blend_radius_m)
    movel([0.203726, -1.353666, -2.590481, -0.768242, 1.570796, 1.774522],accel_mss,speed_ms,0,blend_radius_m)
    movel([0.204454, -1.354137, -2.590166, -0.768086, 1.570796, 1.775250],accel_mss,speed_ms,0,blend_radius_m)
    movel([0.204674, -1.354509, -2.589917, -0.767962, 1.570796, 1.775470],accel_mss,speed_ms,0,blend_radius_m)
    movel([0.205107, -1.355880, -2.588999, -0.767510, 1.570796, 1.775904],accel_mss,speed_ms,0,blend_radius_m)
    movel([0.205169, -1.356670, -2.588469, -0.767250, 1.570796, 1.775965],accel_mss,speed_ms,0,blend_radius_m)
    movel([0.204940, -1.360548, -2.585853, -0.765988, 1.570796, 1.775736],accel_mss,speed_ms,0,blend_radius_m)
    movel([0.204946, -1.360910, -2.585608, -0.765871, 1.570796, 1.775742],accel_mss,speed_ms,0,blend_radius_m)
    movel([0.205235, -1.360658, -2.585779, -0.765952, 1.570796, 1.776031],accel_mss,speed_ms,0,blend_radius_m)
    movel([0.206303, -1.359077, -2.586848, -0.766464, 1.570796, 1.777099],accel_mss,speed_ms,0,blend_radius_m)
    movel([0.206443, -1.358968, -2.586922, -0.766499, 1.570796, 1.777240],accel_mss,speed_ms,0,blend_radius_m)
    movel([0.206778, -1.358969, -2.586921, -0.766499, 1.570796, 1.777575],accel_mss,speed_ms,0,blend_radius_m)
    movel([0.206943, -1.359321, -2.586683, -0.766385, 1.570796, 1.777739],accel_mss,speed_ms,0,blend_radius_m)
    movel([0.206940, -1.360181, -2.586101, -0.766106, 1.570796, 1.777736],accel_mss,speed_ms,0,blend_radius_m)
    movel([0.206733, -1.361999, -2.584869, -0.765521, 1.570796, 1.777529],accel_mss,speed_ms,0,blend_radius_m)
    movel([0.206173, -1.367548, -2.581078, -0.763762, 1.570796, 1.776970],accel_mss,speed_ms,0,blend_radius_m)
    movel([0.205876, -1.373212, -2.577164, -0.762013, 1.570796, 1.776673],accel_mss,speed_ms,0,blend_radius_m)
    movel([0.205845, -1.378146, -2.573717, -0.760526, 1.570796, 1.776641],accel_mss,speed_ms,0,blend_radius_m)
    movel([0.205937, -1.379615, -2.572684, -0.760090, 1.570796, 1.776734],accel_mss,speed_ms,0,blend_radius_m)
    movel([0.206166, -1.381022, -2.571691, -0.759675, 1.570796, 1.776962],accel_mss,speed_ms,0,blend_radius_m)
    movel([0.206613, -1.382309, -2.570781, -0.759299, 1.570796, 1.777409],accel_mss,speed_ms,0,blend_radius_m)
    movel([0.207338, -1.383311, -2.570071, -0.759007, 1.570796, 1.778135],accel_mss,speed_ms,0,blend_radius_m)
    movel([0.208291, -1.383974, -2.569601, -0.758815, 1.570796, 1.779087],accel_mss,speed_ms,0,blend_radius_m)
    movel([0.209418, -1.384254, -2.569401, -0.758734, 1.570796, 1.780215],accel_mss,speed_ms,0,blend_radius_m)
    movel([0.210204, -1.384251, -2.569403, -0.758735, 1.570796, 1.781000],accel_mss,speed_ms,0,blend_radius_m)
    movel([0.211031, -1.384130, -2.569489, -0.758770, 1.570796, 1.781827],accel_mss,speed_ms,0,blend_radius_m)
    movel([0.212970, -1.383552, -2.569900, -0.758937, 1.570796, 1.783766],accel_mss,speed_ms,0,blend_radius_m)
    movel([0.215067, -1.382586, -2.570585, -0.759218, 1.570796, 1.785864],accel_mss,speed_ms,0,blend_radius_m)
    movel([0.217155, -1.381298, -2.571497, -0.759594, 1.570796, 1.787951],accel_mss,speed_ms,0,blend_radius_m)
    movel([0.217790, -1.380896, -2.571781, -0.759713, 1.570796, 1.788586],accel_mss,speed_ms,0,blend_radius_m)
    movel([0.218236, -1.380722, -2.571903, -0.759764, 1.570796, 1.789032],accel_mss,speed_ms,0,blend_radius_m)
    movel([0.218488, -1.380769, -2.571870, -0.759750, 1.570796, 1.789284],accel_mss,speed_ms,0,blend_radius_m)
    movel([0.218570, -1.380999, -2.571707, -0.759682, 1.570796, 1.789366],accel_mss,speed_ms,0,blend_radius_m)
    movel([0.218458, -1.381292, -2.571500, -0.759596, 1.570796, 1.789255],accel_mss,speed_ms,0,blend_radius_m)
    movel([0.218203, -1.381549, -2.571319, -0.759521, 1.570796, 1.789000],accel_mss,speed_ms,0,blend_radius_m)
    movel([0.216603, -1.382597, -2.570577, -0.759215, 1.570796, 1.787399],accel_mss,speed_ms,0,blend_radius_m)
    movel([0.214720, -1.383651, -2.569830, -0.758908, 1.570796, 1.785516],accel_mss,speed_ms,0,blend_radius_m)
    movel([0.212919, -1.384462, -2.569254, -0.758674, 1.570796, 1.783716],accel_mss,speed_ms,0,blend_radius_m)
    movel([0.211601, -1.384887, -2.568951, -0.758551, 1.570796, 1.782398],accel_mss,speed_ms,0,blend_radius_m)
    movel([0.210254, -1.385143, -2.568769, -0.758478, 1.570796, 1.781050],accel_mss,speed_ms,0,blend_radius_m)
    movel([0.209020, -1.385211, -2.568720, -0.758458, 1.570796, 1.779817],accel_mss,speed_ms,0,blend_radius_m)
    movel([0.208049, -1.385072, -2.568819, -0.758498, 1.570796, 1.778845],accel_mss,speed_ms,0,blend_radius_m)
    movel([0.207397, -1.384814, -2.569003, -0.758572, 1.570796, 1.778193],accel_mss,speed_ms,0,blend_radius_m)
    movel([0.206843, -1.384443, -2.569267, -0.758679, 1.570796, 1.777640],accel_mss,speed_ms,0,blend_radius_m)
    movel([0.205895, -1.383330, -2.570057, -0.759001, 1.570796, 1.776692],accel_mss,speed_ms,0,blend_radius_m)
    movel([0.205233, -1.381761, -2.571169, -0.759459, 1.570796, 1.776029],accel_mss,speed_ms,0,blend_radius_m)
    movel([0.204877, -1.379766, -2.572578, -0.760046, 1.570796, 1.775674],accel_mss,speed_ms,0,blend_radius_m)
    movel([0.204766, -1.377269, -2.574332, -0.760788, 1.570796, 1.775562],accel_mss,speed_ms,0,blend_radius_m)
    movel([0.204821, -1.373582, -2.576907, -0.761900, 1.570796, 1.775617],accel_mss,speed_ms,0,blend_radius_m)
    movel([0.205008, -1.369497, -2.579736, -0.763155, 1.570796, 1.775804],accel_mss,speed_ms,0,blend_radius_m)
    movel([0.205313, -1.365632, -2.582392, -0.764365, 1.570796, 1.776109],accel_mss,speed_ms,0,blend_radius_m)
    movel([0.205666, -1.361861, -2.584963, -0.765565, 1.570796, 1.776463],accel_mss,speed_ms,0,blend_radius_m)
    movel([0.205643, -1.361723, -2.585056, -0.765609, 1.570796, 1.776439],accel_mss,speed_ms,0,blend_radius_m)
    movel([0.205470, -1.361828, -2.584986, -0.765576, 1.570796, 1.776266],accel_mss,speed_ms,0,blend_radius_m)
    movel([0.205173, -1.362084, -2.584812, -0.765494, 1.570796, 1.775969],accel_mss,speed_ms,0,blend_radius_m)
    movel([0.204799, -1.362215, -2.584722, -0.765451, 1.570796, 1.775596],accel_mss,speed_ms,0,blend_radius_m)
    movel([0.204420, -1.362190, -2.584739, -0.765459, 1.570796, 1.775217],accel_mss,speed_ms,0,blend_radius_m)
    movel([0.204117, -1.362013, -2.584860, -0.765516, 1.570796, 1.774914],accel_mss,speed_ms,0,blend_radius_m)
    movel([0.203979, -1.361774, -2.585022, -0.765593, 1.570796, 1.774776],accel_mss,speed_ms,0,blend_radius_m)
    movel([0.203910, -1.360786, -2.585692, -0.765911, 1.570796, 1.774707],accel_mss,speed_ms,0,blend_radius_m)
    movel([0.203975, -1.359813, -2.586351, -0.766225, 1.570796, 1.774771],accel_mss,speed_ms,0,blend_radius_m)
    movel([0.204080, -1.357514, -2.587902, -0.766973, 1.570796, 1.774877],accel_mss,speed_ms,0,blend_radius_m)
    movel([0.203938, -1.355959, -2.588946, -0.767484, 1.570796, 1.774734],accel_mss,speed_ms,0,blend_radius_m)
    movel([0.203557, -1.354980, -2.589602, -0.767807, 1.570796, 1.774353],accel_mss,speed_ms,0,blend_radius_m)
    movel([0.203287, -1.354696, -2.589793, -0.767901, 1.570796, 1.774083],accel_mss,speed_ms,0,blend_radius_m)
    movel([0.202556, -1.354463, -2.589948, -0.767978, 1.570796, 1.773352],accel_mss,speed_ms,0,blend_radius_m)
    movel([0.202308, -1.354479, -2.589937, -0.767972, 1.570796, 1.773104],accel_mss,speed_ms,0,blend_radius_m)
    movel([0.201509, -1.354860, -2.589683, -0.767846, 1.570796, 1.772306],accel_mss,speed_ms,0,blend_radius_m)
    movel([0.200401, -1.355577, -2.589203, -0.767610, 1.570796, 1.771198],accel_mss,speed_ms,0,blend_radius_m)
    movel([0.199384, -1.356426, -2.588633, -0.767330, 1.570796, 1.770180],accel_mss,speed_ms,0,blend_radius_m)
    movel([0.196714, -1.359160, -2.586792, -0.766437, 1.570796, 1.767511],accel_mss,speed_ms,0,blend_radius_m)
    movel([0.194140, -1.362290, -2.584672, -0.765428, 1.570796, 1.764936],accel_mss,speed_ms,0,blend_radius_m)
    movel([0.193117, -1.363743, -2.583682, -0.764963, 1.570796, 1.763913],accel_mss,speed_ms,0,blend_radius_m)
    movel([0.192215, -1.365218, -2.582675, -0.764495, 1.570796, 1.763011],accel_mss,speed_ms,0,blend_radius_m)
    movel([0.190820, -1.367872, -2.580856, -0.763661, 1.570796, 1.761616],accel_mss,speed_ms,0,blend_radius_m)
    movel([0.189760, -1.370335, -2.579158, -0.762896, 1.570796, 1.760557],accel_mss,speed_ms,0,blend_radius_m)
    movel([0.188929, -1.372876, -2.577398, -0.762116, 1.570796, 1.759725],accel_mss,speed_ms,0,blend_radius_m)
    movel([0.188225, -1.375765, -2.575385, -0.761239, 1.570796, 1.759022],accel_mss,speed_ms,0,blend_radius_m)
    movel([0.187720, -1.378680, -2.573342, -0.760367, 1.570796, 1.758516],accel_mss,speed_ms,0,blend_radius_m)
    movel([0.187446, -1.381521, -2.571339, -0.759529, 1.570796, 1.758242],accel_mss,speed_ms,0,blend_radius_m)
    movel([0.187392, -1.384296, -2.569371, -0.758722, 1.570796, 1.758188],accel_mss,speed_ms,0,blend_radius_m)
    movel([0.187560, -1.386978, -2.567459, -0.757952, 1.570796, 1.758356],accel_mss,speed_ms,0,blend_radius_m)
    movel([0.187949, -1.389597, -2.565582, -0.757210, 1.570796, 1.758745],accel_mss,speed_ms,0,blend_radius_m)
    movel([0.188554, -1.392101, -2.563778, -0.756510, 1.570796, 1.759350],accel_mss,speed_ms,0,blend_radius_m)
    movel([0.189381, -1.394543, -2.562009, -0.755837, 1.570796, 1.760178],accel_mss,speed_ms,0,blend_radius_m)
    movel([0.190402, -1.396861, -2.560323, -0.755205, 1.570796, 1.761199],accel_mss,speed_ms,0,blend_radius_m)
    movel([0.191484, -1.398761, -2.558935, -0.754693, 1.570796, 1.762280],accel_mss,speed_ms,0,blend_radius_m)
    movel([0.192768, -1.400509, -2.557653, -0.754227, 1.570796, 1.763565],accel_mss,speed_ms,0,blend_radius_m)
    movel([0.194072, -1.401803, -2.556701, -0.753885, 1.570796, 1.764869],accel_mss,speed_ms,0,blend_radius_m)
    movel([0.195629, -1.402859, -2.555922, -0.753608, 1.570796, 1.766426],accel_mss,speed_ms,0,blend_radius_m)
    movel([0.197217, -1.403539, -2.555420, -0.753430, 1.570796, 1.768014],accel_mss,speed_ms,0,blend_radius_m)
    movel([0.199012, -1.403941, -2.555123, -0.753325, 1.570796, 1.769808],accel_mss,speed_ms,0,blend_radius_m)
    movel([0.200910, -1.404036, -2.555053, -0.753301, 1.570796, 1.771707],accel_mss,speed_ms,0,blend_radius_m)
    movel([0.202935, -1.403817, -2.555215, -0.753358, 1.570796, 1.773731],accel_mss,speed_ms,0,blend_radius_m)
    movel([0.204801, -1.403351, -2.555559, -0.753479, 1.570796, 1.775597],accel_mss,speed_ms,0,blend_radius_m)
    movel([0.206681, -1.402623, -2.556096, -0.753669, 1.570796, 1.777477],accel_mss,speed_ms,0,blend_radius_m)
    movel([0.208573, -1.401639, -2.556822, -0.753928, 1.570796, 1.779369],accel_mss,speed_ms,0,blend_radius_m)
    movel([0.210385, -1.400448, -2.557698, -0.754244, 1.570796, 1.781182],accel_mss,speed_ms,0,blend_radius_m)
    movel([0.212328, -1.398895, -2.558837, -0.754658, 1.570796, 1.783124],accel_mss,speed_ms,0,blend_radius_m)
    movel([0.214124, -1.397193, -2.560080, -0.755115, 1.570796, 1.784920],accel_mss,speed_ms,0,blend_radius_m)
    movel([0.216116, -1.395029, -2.561657, -0.755704, 1.570796, 1.786912],accel_mss,speed_ms,0,blend_radius_m)
    movel([0.219248, -1.391251, -2.564391, -0.756747, 1.570796, 1.790045],accel_mss,speed_ms,0,blend_radius_m)
    movel([0.220263, -1.390231, -2.565126, -0.757032, 1.570796, 1.791060],accel_mss,speed_ms,0,blend_radius_m)
    movel([0.221225, -1.389519, -2.565638, -0.757232, 1.570796, 1.792021],accel_mss,speed_ms,0,blend_radius_m)
    movel([0.222300, -1.388971, -2.566032, -0.757387, 1.570796, 1.793096],accel_mss,speed_ms,0,blend_radius_m)
    movel([0.223237, -1.388662, -2.566253, -0.757474, 1.570796, 1.794034],accel_mss,speed_ms,0,blend_radius_m)
    movel([0.224148, -1.388517, -2.566357, -0.757515, 1.570796, 1.794944],accel_mss,speed_ms,0,blend_radius_m)
    movel([0.224981, -1.388543, -2.566339, -0.757508, 1.570796, 1.795777],accel_mss,speed_ms,0,blend_radius_m)
    movel([0.225715, -1.388738, -2.566199, -0.757452, 1.570796, 1.796511],accel_mss,speed_ms,0,blend_radius_m)
    movel([0.226396, -1.389124, -2.565922, -0.757343, 1.570796, 1.797192],accel_mss,speed_ms,0,blend_radius_m)
    movel([0.226932, -1.389655, -2.565540, -0.757194, 1.570796, 1.797728],accel_mss,speed_ms,0,blend_radius_m)
    movel([0.227406, -1.390402, -2.565003, -0.756984, 1.570796, 1.798202],accel_mss,speed_ms,0,blend_radius_m)
    movel([0.227756, -1.391229, -2.564407, -0.756753, 1.570796, 1.798553],accel_mss,speed_ms,0,blend_radius_m)
    movel([0.228419, -1.394028, -2.562383, -0.755978, 1.570796, 1.799215],accel_mss,speed_ms,0,blend_radius_m)
    movel([0.228644, -1.395601, -2.561241, -0.755547, 1.570796, 1.799440],accel_mss,speed_ms,0,blend_radius_m)
    movel([0.228757, -1.397980, -2.559506, -0.754903, 1.570796, 1.799554],accel_mss,speed_ms,0,blend_radius_m)
    movel([0.228704, -1.398816, -2.558895, -0.754679, 1.570796, 1.799501],accel_mss,speed_ms,0,blend_radius_m)
    movel([0.228321, -1.400957, -2.557324, -0.754109, 1.570796, 1.799117],accel_mss,speed_ms,0,blend_radius_m)
    movel([0.227895, -1.402658, -2.556070, -0.753660, 1.570796, 1.798691],accel_mss,speed_ms,0,blend_radius_m)
    movel([0.227411, -1.404077, -2.555022, -0.753290, 1.570796, 1.798208],accel_mss,speed_ms,0,blend_radius_m)
    movel([0.226774, -1.405476, -2.553986, -0.752927, 1.570796, 1.797570],accel_mss,speed_ms,0,blend_radius_m)
    movel([0.225879, -1.407112, -2.552770, -0.752507, 1.570796, 1.796675],accel_mss,speed_ms,0,blend_radius_m)
    movel([0.224743, -1.408910, -2.551429, -0.752050, 1.570796, 1.795539],accel_mss,speed_ms,0,blend_radius_m)
    movel([0.223465, -1.410663, -2.550117, -0.751609, 1.570796, 1.794261],accel_mss,speed_ms,0,blend_radius_m)
    movel([0.221708, -1.412851, -2.548474, -0.751064, 1.570796, 1.792504],accel_mss,speed_ms,0,blend_radius_m)
    movel([0.217862, -1.417214, -2.545174, -0.750000, 1.570796, 1.788658],accel_mss,speed_ms,0,blend_radius_m)
    movel([0.215781, -1.419381, -2.543526, -0.749482, 1.570796, 1.786577],accel_mss,speed_ms,0,blend_radius_m)
    movel([0.213809, -1.421307, -2.542054, -0.749028, 1.570796, 1.784605],accel_mss,speed_ms,0,blend_radius_m)
    movel([0.211760, -1.423165, -2.540629, -0.748595, 1.570796, 1.782557],accel_mss,speed_ms,0,blend_radius_m)
    movel([0.209118, -1.425477, -2.538849, -0.748063, 1.570796, 1.779915],accel_mss,speed_ms,0,blend_radius_m)
    movel([0.209901, -1.425337, -2.538957, -0.748095, 1.570796, 1.780698],accel_mss,speed_ms,0,blend_radius_m)
    movel([0.210596, -1.425288, -2.538995, -0.748106, 1.570796, 1.781392],accel_mss,speed_ms,0,blend_radius_m)
    movel([0.210823, -1.425356, -2.538942, -0.748091, 1.570796, 1.781620],accel_mss,speed_ms,0,blend_radius_m)
    movel([0.211213, -1.425683, -2.538690, -0.748016, 1.570796, 1.782009],accel_mss,speed_ms,0,blend_radius_m)
    movel([0.211285, -1.425865, -2.538550, -0.747975, 1.570796, 1.782082],accel_mss,speed_ms,0,blend_radius_m)
    movel([0.211176, -1.426473, -2.538079, -0.747836, 1.570796, 1.781972],accel_mss,speed_ms,0,blend_radius_m)
    movel([0.210961, -1.427154, -2.537552, -0.747682, 1.570796, 1.781757],accel_mss,speed_ms,0,blend_radius_m)
    movel([0.213179, -1.426802, -2.537825, -0.747762, 1.570796, 1.783975],accel_mss,speed_ms,0,blend_radius_m)
    movel([0.213716, -1.426647, -2.537945, -0.747797, 1.570796, 1.784513],accel_mss,speed_ms,0,blend_radius_m)
    movel([0.216064, -1.425787, -2.538609, -0.747992, 1.570796, 1.786860],accel_mss,speed_ms,0,blend_radius_m)
    movel([0.216496, -1.425720, -2.538661, -0.748008, 1.570796, 1.787292],accel_mss,speed_ms,0,blend_radius_m)
    movel([0.216889, -1.425755, -2.538634, -0.748000, 1.570796, 1.787686],accel_mss,speed_ms,0,blend_radius_m)
    movel([0.217292, -1.425982, -2.538459, -0.747948, 1.570796, 1.788088],accel_mss,speed_ms,0,blend_radius_m)
    movel([0.217466, -1.426389, -2.538145, -0.747855, 1.570796, 1.788262],accel_mss,speed_ms,0,blend_radius_m)
    movel([0.217419, -1.427077, -2.537612, -0.747700, 1.570796, 1.788216],accel_mss,speed_ms,0,blend_radius_m)
    movel([0.216847, -1.429358, -2.535842, -0.747188, 1.570796, 1.787643],accel_mss,speed_ms,0,blend_radius_m)
    movel([0.216815, -1.429644, -2.535620, -0.747125, 1.570796, 1.787611],accel_mss,speed_ms,0,blend_radius_m)
    movel([0.217302, -1.429525, -2.535712, -0.747151, 1.570796, 1.788098],accel_mss,speed_ms,0,blend_radius_m)
    movel([0.220607, -1.427262, -2.537469, -0.747658, 1.570796, 1.791403],accel_mss,speed_ms,0,blend_radius_m)
    movel([0.222012, -1.426212, -2.538281, -0.747896, 1.570796, 1.792808],accel_mss,speed_ms,0,blend_radius_m)
    movel([0.225160, -1.423547, -2.540336, -0.748506, 1.570796, 1.795957],accel_mss,speed_ms,0,blend_radius_m)
    movel([0.227121, -1.421733, -2.541728, -0.748928, 1.570796, 1.797917],accel_mss,speed_ms,0,blend_radius_m)
    movel([0.234533, -1.414542, -2.547198, -0.750649, 1.570796, 1.805330],accel_mss,speed_ms,0,blend_radius_m)
    movel([0.238371, -1.410652, -2.550126, -0.751612, 1.570796, 1.809167],accel_mss,speed_ms,0,blend_radius_m)
    movel([0.241467, -1.407330, -2.552607, -0.752451, 1.570796, 1.812264],accel_mss,speed_ms,0,blend_radius_m)
    movel([0.244047, -1.404331, -2.554834, -0.753224, 1.570796, 1.814843],accel_mss,speed_ms,0,blend_radius_m)
    movel([0.248637, -1.398374, -2.559218, -0.754797, 1.570796, 1.819433],accel_mss,speed_ms,0,blend_radius_m)
    movel([0.251323, -1.394759, -2.561852, -0.755777, 1.570796, 1.822119],accel_mss,speed_ms,0,blend_radius_m)
    movel([0.253903, -1.390958, -2.564602, -0.756828, 1.570796, 1.824700],accel_mss,speed_ms,0,blend_radius_m)
    movel([0.254663, -1.389666, -2.565532, -0.757191, 1.570796, 1.825460],accel_mss,speed_ms,0,blend_radius_m)
    movel([0.255148, -1.388711, -2.566218, -0.757460, 1.570796, 1.825945],accel_mss,speed_ms,0,blend_radius_m)
    movel([0.255131, -1.388396, -2.566444, -0.757549, 1.570796, 1.825927],accel_mss,speed_ms,0,blend_radius_m)
